// TwinCAT 3 PLC project PLC_STATE_DRIVE
// Title: PLC_STATE_DRIVE
// Author: D. Hauer
// ProjectVersion: 01.00.10
// Description: MC-PtP, NCI, Camming cyclic execution layer for motion commands
// ProgramVersion: 3.1.4024.0
// libraries:
//   Tc2_MC2, * (Beckhoff Automation GmbH)
//   Tc2_MC2_Camming, * (Beckhoff Automation GmbH)
//   Tc2_MC2_Drive, * (Beckhoff Automation GmbH)
//   Tc2_NC, * (Beckhoff Automation GmbH)
//   Tc2_Standard, * (Beckhoff Automation GmbH)
//   Tc2_System, * (Beckhoff Automation GmbH)
//   Tc2_Utilities, * (Beckhoff Automation GmbH)
//   Tc3_Module, * (Beckhoff Automation GmbH)
//   Tc2_NCI,3.3.15.0,Beckhoff Automation GmbH
//   Tc2_PlcInterpolation,3.3.18.0,Beckhoff Automation GmbH
// project tree:
//   / CAM.TcPOU, NCI.TcPOU, MAIN.TcPOU, PlcTask.TcTTO, Visualization Manager.TcVMO (not stored)
//   CAM/ FB_CamAxis.TcPOU, FB_CamCtrl.TcPOU, I_Cam_Ctrl.TcIO
//   CAM/types/ ST_CAM_CTRL.TcDUT, ST_CAM_DATA.TcDUT, ST_CAM_INFO.TcDUT, ST_CAM_READ_VALUES_PARAMETER.TcDUT (not stored), ST_CAM_STATE.TcDUT, ST_CAM_OPTIONS.TcDUT, ST_CAM_SCALING_DATA.TcDUT, ST_MOTION_FUNCTION.TcDUT (not stored), ST_MOTION_FUNCTION_POINT.TcDUT (not stored)
//   MAPPING/ MAPPING_in.TcPOU, MAPPING_out.TcPOU
//   MAPPING/types/ U_AXIS_CTRL.TcDUT (not stored), U_AXIS_NC_PARAMETER_WRT.TcDUT (not stored), U_AXIS_HOMING.TcDUT (not stored), U_AXIS_MOTION_OPTIONS.TcDUT (not stored), U_AXIS_MOVE_DATA.TcDUT (not stored), U_AXIS_GEAR_IN.TcDUT (not stored), U_AXIS_NC_PARAMETER_RD.TcDUT (not stored), U_AXIS_STATE.TcDUT (not stored), U_AXIS_INFO.TcDUT (not stored)
//   NCI/ FB_NciChannelCtrl.TcPOU, FB_NciChannel.TcPOU, I_NciChannel.TcIO, I_Nci_Ctrl.TcIO
//   NCI/types/ E_NCI_CTRL.TcDUT, E_NCI_CHANNEL_ERROR.TcDUT (not stored), E_NCI_STATE.TcDUT, E_NCI_INTERPRETER_STATE.TcDUT (not stored), ST_3D_Group.TcDUT (not stored), ST_CTRL_NCI.TcDUT, ST_NCI_M_FUNC.TcDUT, ST_Index_Group.TcDUT (not stored), ST_Interface_Group.TcDUT (not stored), ST_NciChannel_Ref.TcDUT (not stored), ST_R_Parameter.TcDUT, ST_STATE_NCI.TcDUT
//   NC_PTP/ FB_McAxisCtrl.TcPOU, FB_McAxis.TcPOU, I_McAxis.TcIO
//   NC_PTP/types/axis/ E_AxisEncoderType.TcDUT (not stored), ST_HomeParams.TcDUT
//   NC_PTP/types/control/ E_AXIS_CTRL.TcDUT, E_AXIS_STATE.TcDUT, ST_AXIS_CTRL.TcDUT, ST_AXIS_INFO.TcDUT, ST_AXIS_STATE.TcDUT, ST_GEAR_IN.TcDUT, ST_HOMING.TcDUT (not stored), ST_MOTION_OPTIONS.TcDUT, ST_MOVE_DATA.TcDUT (not stored), ST_NC_PARAMETER.TcDUT (not stored)
//   _DUT/ E_CHECK_STATE.TcDUT, E_PROGRESS.TcDUT
//   _GVL/ GlobalTextList.TcGTLO, GVL_AXIS.TcGVL, GVL_CAM.TcGVL, GVL_MSG.TcGVL, GVL_NCI.TcGVL, PLC_CONSTANT.TcGVL, PLC_VERSION.TcGVL
//   _MSG/ fb_LocalTime.TcPOU (not stored), f_MessageSet.TcPOU, MessageData.TcPOU, T_MESSAGE_LIST.TcVIS
//   _MSG/types/ e_Device.TcDUT, E_MessageType.TcDUT, E_MESSAGE_STATE.TcDUT (not stored), e_Subdevice.TcDUT, ST_Message.TcDUT
//   _UML/ CD_AXIS_ACCESS.TcCD (not stored) (excluded from build), CD_CAM_ACCESS.TcCD (not stored) (excluded from build)

CONFIGURATION PLC_STATE_DRIVE
    RESOURCE PLC ON TwinCAT3
        TASK PlcTask(INTERVAL := T#10ms, PRIORITY := 20);
        PROGRAM MAPPING_in WITH PlcTask : MAPPING_in;
        PROGRAM LEGACY WITH PlcTask : LEGACY;
        PROGRAM MAIN WITH PlcTask : MAIN;
        PROGRAM NCI WITH PlcTask : NCI;
        PROGRAM CAM WITH PlcTask : CAM;
        PROGRAM MAPPING_out WITH PlcTask : MAPPING_out;
    END_RESOURCE
END_CONFIGURATION

// ---- CAM/types/ST_CAM_CTRL.TcDUT
{attribute 'pack_mode' := '2'}
TYPE ST_CAM_CTRL :
STRUCT
  eCtrl               : E_AXIS_CTRL;    // commanded axis function
END_STRUCT
END_TYPE

// ---- CAM/types/ST_CAM_DATA.TcDUT
{attribute 'pack_mode' := '2'}
TYPE ST_CAM_DATA :
STRUCT
  // MC_CamInfo_V2 parameters
  bAtMasterPosition       : BIT;    // If AtMasterPosition is TRUE, the data related to the specified MasterPosition is determined. Otherwise the data refers to the current master position.
  nMasterIndex            : UINT;   // Index in GVL_AXIS.AxisRef[nMasterIndex]

  rMasterPosition         : LREAL;  // Master position to which the data that is determined refers. This input parameter is not necessary if AtMasterPosition is FALSE.
  rActivationPosition     : LREAL;
  nActivationMode         : UINT;
  nCamTableId             : UDINT;  // For multi-cam plate coupling, the CamTableId also has to be transferred explicitly. If a single cam plate is involved in the coupling, the CamTableId can be set to 0.
  nPointId                : UDINT;
  nNumPoints              : UDINT;  // 0 = full motion function size

  stCamScalingData        : ST_CAM_SCALING_DATA;
  stOptions               : ST_CAM_OPTIONS;
END_STRUCT
END_TYPE

// ---- CAM/types/ST_CAM_INFO.TcDUT
{attribute 'pack_mode' := '2'}
TYPE ST_CAM_INFO :
STRUCT
  bError              : BIT;
  wCamCouplingState   : ARRAY[0..7] OF WORD;
  nCamCouplingTableId : ARRAY[0..7] OF UINT;

  nNumPointsRead      : UDINT;
END_STRUCT
END_TYPE

// ---- CAM/types/ST_CAM_STATE.TcDUT
{attribute 'pack_mode' := '2'}
TYPE ST_CAM_STATE :
STRUCT
  nNumPointsRead          : UDINT;

END_STRUCT
END_TYPE

// ---- CAM/types/ST_CAM_OPTIONS.TcDUT
{attribute 'pack_mode' := '2'}
TYPE ST_CAM_OPTIONS :
STRUCT
  nInterpolationType      : UINT;
  nCamOperationMode       : UINT;
  nReferenceCamTableId    : UDINT;
END_STRUCT
END_TYPE

// ---- CAM/types/ST_CAM_SCALING_DATA.TcDUT
{attribute 'pack_mode' := '2'}
TYPE ST_CAM_SCALING_DATA :
STRUCT
  // scaling of X-axis (Master) of the CAM
  nMasterScalingMode      : UINT;
  bMasterRelative         : BOOL;
  rMasterOffset           : LREAL;
  rMasterScaling          : LREAL := 1.0;

  // scaling of Y-axis (Slave) of CAM
  nSlaveScalingMode       : UINT;
  bSlaveRelative          : BOOL;
  rSlaveOffset            : LREAL;
  rSlaveScaling           : LREAL := 1.0;
END_STRUCT
END_TYPE

// ---- NCI/types/E_NCI_CTRL.TcDUT
{attribute 'qualified_only'}
{attribute 'to_string'}
TYPE E_NCI_CTRL :
(
  NO_NCI            := -10,
  NO_AXIS_GROUP     := -2,
  NO_AXIS_INDEX     := -1,
  NO_INIT,
  INIT,
  IDLE,
  RESET,
  LOAD_PROG,
  FEED_TABLE,
  BUILD_GROUP,
  CLEAR_GROUP,

  START         := 10,
  STOP,
  STO_STOP,
  RESTART_STEP_ON,

  M_FUNC_QUIT   := 20,

  READ_R_PARA   := 30,
  WRITE_R_PARA  := 40,

  CMD_BUSY      := 100,
  CMD_DONE      := 1000,
  CMD_ERROR     := 9000
)DINT;
END_TYPE

// ---- NCI/types/E_NCI_STATE.TcDUT
{attribute 'qualified_only'}
//{attribute 'strict'}
{attribute 'to_string'}
TYPE E_NCI_STATE :
(
  NO_NCI            := -10,
  NO_AXIS_GROUP     := -2,
  NO_AXIS_INDEX     := -1,
  NO_INIT,
  INIT,
  IDLE,
  RESET,
  LOAD_PROG,
  FEED_TABLE,
  BUILD_GROUP,
  CLEAR_GROUP,

  START         := 10,
  STOP,
  STO_STOP,
  RESTART_STEP_ON,

  M_FUNC_QUIT   := 20,

  READ_R_PARA   := 30,
  WRITE_R_PARA  := 40

)DINT;
END_TYPE

// ---- NCI/types/ST_CTRL_NCI.TcDUT
{attribute 'pack_mode' := '2'}
TYPE ST_CTRL_NCI :
STRUCT
  eCmd        : E_NCI_CTRL := E_NCI_CTRL.INIT;
  rOverride   : REAL := 47.11;

END_STRUCT
END_TYPE

// ---- NCI/types/ST_NCI_M_FUNC.TcDUT
{attribute 'pack_mode' := '2'}
TYPE ST_NCI_M_FUNC :
STRUCT
  FastMFuncMask   : ARRAY [1..5] OF DWORD;
  HskMFuncNo      : UINT;
  HskMFuncReq     : WORD;
  HFuncValue      : UDINT; 
END_STRUCT
END_TYPE

// ---- NCI/types/ST_R_Parameter.TcDUT
{attribute 'pack_mode' := '2'}
TYPE ST_R_Parameter :
STRUCT
  _nStart               : DINT := 901;
  _nCount               : DINT :=   4;
  _rRParamsWrite        : ARRAY[0..MAX_R_PARA] OF LREAL := [11.11, 22.22, 33.33, 456.22];
  _rRParamsRead         : ARRAY[0..MAX_R_PARA] OF LREAL;
END_STRUCT
END_TYPE

// ---- NCI/types/ST_STATE_NCI.TcDUT
{attribute 'pack_mode' := '2'}
TYPE ST_STATE_NCI :
STRUCT
  eState        : E_NCI_STATE; // eCmd with offsets E_PROGRESS

  bMFuncReq     : BIT;  // M function request is active from channel

  nMFunc        : WORD; // number of active M function

  nItpState     : UINT; 
                         (*  Interpreter Operation State:
                            0  = Init failed
                            1  = Idle
                            2  = Ready
                            3  = Started
                            4  = Scanning
                            5  = Running
                            6  = Stay running
                            7  = Write table
                            8  = Search line
                            9  = End
                            10 = Single Step
                            11 = Aborting
                            12 = Aborted
                            13 = Fault
                            14 = Reset
                            15 = Stop
                            16 = Wait function
                            17 = Flush buffers
                          *) 

  rAxisOverride : REAL; // active override in cyclic NCI interface

END_STRUCT
END_TYPE

// ---- NC_PTP/types/axis/ST_HomeParams.TcDUT
TYPE ST_HomeParams :
STRUCT
  Position              : LREAL;
  HomingMode            : Tc2_MC2.MC_HomingMode;
  Options               : Tc2_MC2.ST_HomingOptions;

  InvertHomeSensor      : BIT := FALSE;   //Set to true,  NormallyClosed home sensor
  SimulateHomeSensor    : BIT := FALSE;   //Set to true,  homed on encoder index only. The homing methode 'hardware sync' must be used then.

  UseLimitMin           : BIT := TRUE;    //Set to false, no negative limit sensor.

  InvertLimitMin        : BIT := FALSE;   //Set to true,  NC negative limit sensor
  HomeOnLimitMin        : BIT := FALSE;   //Set to true,  homed on negative limit sensor 

  UseLimitMax           : BIT := TRUE;    //Set to false, no positive limit sensor.

  InvertLimitMax        : BIT := FALSE;   //Set to true,  NC positive limit sensor
  HomeOnLimitMax        : BIT := FALSE;   //Set to true,  homed on positive limit sensor 
  
  // It is not allowed to use more than 1 of the 3 switches: SimulateHomeSensor, HomeOnLimitMin, HomeOnLimitMax
  
END_STRUCT
END_TYPE

// ---- NC_PTP/types/control/E_AXIS_CTRL.TcDUT
{attribute 'qualified_only'}
{attribute 'strict'}
{attribute 'to_string'}
TYPE E_AXIS_CTRL :
(
  AXIS_NULL,   // null command
  AXIS_INIT,
  AXIS_DISABLE,
  AXIS_ENABLE,

  AXIS_IDLE     := 10, // clear axis and enable
  AXIS_HOME,
  AXIS_MOVE_POS,
  AXIS_MOVE_VELO,
  AXIS_HALT,
  AXIS_STOP,

  AXIS_RESET              := 19,
  AXIS_STARTUP            := 20,

  AXIS_MOVE_BUFFER        := 30,
  AXIS_MOVE_BUFFER_VELO,

  AXIS_PARAMETER_READ     := 40, // command for reading and writing parameter
  AXIS_PARAMETER_WRITE,
  AXIS_PARAMETER_WRITE_PERSISTENT,


  AXIS_GEAR_IN            := 50,
  AXIS_GEAR_OUT,
  AXIS_GEAR_IN_MULTIMASTER,

  CAM_INIT                := 60,
  CAM_IN,
  CAM_SCALING,
  CAM_INFO,
  CAM_RD_MOTION_FUNCTION,
  CAM_RD_MOTION_FUNCTION_POINT,
  CAM_RD_MOTION_FUNCTIONS_VALUES,
  CAM_WRT_MOTION_FUNCTION,
  CAM_WRT_MOTION_FUNCTION_POINT

)UINT;
END_TYPE

// ---- NC_PTP/types/control/E_AXIS_STATE.TcDUT
{attribute 'qualified_only'}
{attribute 'to_string'}
TYPE E_AXIS_STATE :
(
  AXIS_NULL,   // null reaction to command
  AXIS_INIT,
  AXIS_DISABLE,
  AXIS_ENABLE,

  AXIS_NO_INIT  := 9,
  
  AXIS_IDLE     := 10, // clear axis and enable
  AXIS_HOME,
  AXIS_MOVE_POS,
  AXIS_MOVE_VELO,
  AXIS_HALT,
  AXIS_STOP,

  AXIS_RESET              := 19,
  AXIS_STARTUP            := 20,

  AXIS_MOVE_BUFFER        := 30,
  AXIS_MOVE_BUFFER_VELO,

  AXIS_PARAMETER_READ     := 40, // command for reading and writing parameter
  AXIS_PARAMETER_WRITE,
  AXIS_PARAMETER_WRITE_PERSISTENT,


  AXIS_GEAR_IN            := 50,
  AXIS_GEAR_OUT,
  AXIS_GEAR_IN_MULTIMASTER,

  CAM_INIT                := 60,
  CAM_IN,
  CAM_SCALING,
  CAM_INFO,
  CAM_RD_MOTION_FUNCTION,
  CAM_RD_MOTION_FUNCTION_POINT,
  CAM_RD_MOTION_FUNCTIONS_VALUES,
  CAM_WRT_MOTION_FUNCTION,
  CAM_WRT_MOTION_FUNCTION_POINT

)UINT;
END_TYPE

// ---- NC_PTP/types/control/ST_AXIS_CTRL.TcDUT
{attribute 'pack_mode' := '2'}
TYPE ST_AXIS_CTRL :
STRUCT
  eCtrl               : E_AXIS_CTRL;    // commanded axis function
  eProgress           : E_PROGRESS;     // progress command for synced functions
END_STRUCT
END_TYPE

// ---- NC_PTP/types/control/ST_AXIS_INFO.TcDUT
{attribute 'pack_mode' := '2'}
TYPE ST_AXIS_INFO :
STRUCT
  bEnabled    : BIT; // Enabled: check if ControlLoop is closed and active
  bReferenced : BIT; // Axis homing bit
  bReady      : BIT; // enabled & NOT bError & no Axis Function requested
  bBusy       : BIT; // axis function requested or active
  bError      : BIT;
  bTimeout    : BIT; // for move cmds or switching drive on timeout
  bInTarget   : BIT; // ActPos = SetPos --> position check is done with configured window in NC
  bStandstill : BIT; // No Error and NOT moving
 
  nErrorId            : UDINT;

  rActPos             : LREAL;
  rActVelo            : LREAL;
  rPosDiff            : LREAL;

  dwCoupleState       : DWORD;   // cyclic information about axis couple state
END_STRUCT
END_TYPE

// ---- NC_PTP/types/control/ST_AXIS_STATE.TcDUT
{attribute 'pack_mode' := '2'}
TYPE ST_AXIS_STATE :
STRUCT
  eState        : E_AXIS_STATE; // mirror the requested command + E_PROGRESS
  eAxisEncoder  : E_AxisEncoderType;
END_STRUCT
END_TYPE

// ---- NC_PTP/types/control/ST_GEAR_IN.TcDUT
{attribute 'pack_mode' := '2'}
TYPE ST_GEAR_IN :
STRUCT  
  nAxisIndexMaster    : ARRAY [1..4] OF BYTE; // Index of Master1-4
  rGearRatio          : ARRAY [1..4] OF REAL; 
  Acceleration        : REAL;
  Deceleration        : REAL;
  Jerk                : REAL;  
END_STRUCT
END_TYPE

// ---- NC_PTP/types/control/ST_MOTION_OPTIONS.TcDUT
{attribute 'pack_mode' := '2'}
TYPE ST_MOTION_OPTIONS :
STRUCT
  eBufferMode   : Tc2_MC2.MC_BufferMode;

END_STRUCT
END_TYPE

// ---- _DUT/E_CHECK_STATE.TcDUT
{attribute 'qualified_only'}
{attribute 'strict'}
{attribute 'to_string'}
TYPE E_CHECK_STATE :
(
  CHECK_INIT,
  AXIS_INDEX_OUT_OF_RANGE         :=  10,

	AXIS_REF_POINTER_INVALID        := 100,
  AXIS_CTRL_POINTER_INVALID,
  AXIS_STATE_POINTER_INVALID,
  AXIS_INFO_POINTER_INVALID,
  AXIS_DATA_POINTER_INVALID,
  AXIS_NC_PARAMETER_POINTER_INVALID,
  AXIS_HOME_PARAMETER_POINTER_INVALID,
  AXIS_GEAR_IN_PARAMETER_POINTER_INVALID,
  AXIS_GEAR_IN_MULTIMASTER_POINTER_INVALID,
  AXIS_MOTION_OPTIONS_POINTER_INVALID,

  NCI_NOT_ACTIVATED               := 200,
  NCI_CHANNEL_REF_POINTER_INVALID,
  NCI_AXIS_CONFIG_POINTER_INVALID,
  NCI_MCS_AXIS_POINTER_INVALID,
  NCI_AUX_AXIS_POINTER_INVALID,
  NCI_CTRL_POINTER_INVALID,
  NCI_STATE_POINTER_INVALID,
  NCI_R_PARAMETER_READ_POINTER_INVALID,
  NCI_R_PARAMETER_wRITE_POINTER_INVALID,
  NCI_M_FUNC_POINTER_INVALID,

  CAM_NOT_ACTIVATED               := 300,
  CAM_SLAVE_AXIS_REF_INVALID,
  CAM_SLAVE_ITF_MC_AXIS_INVALID,
  CAM_MASTER_AXIS_REF_INVALID,
  CAM_MOTION_FUNCTION_POINTER_INVALID,
  CAM_MOTION_FUNCTION_POINT_POINTER_INVALID,

  CHECK_DONE                      := 10000
  
)UINT;
END_TYPE

// ---- _DUT/E_PROGRESS.TcDUT
{attribute 'qualified_only'}
//{attribute 'strict'}
{attribute 'to_string'}
TYPE E_PROGRESS :
(
  // progress is used in project to mirror state of requested command/function
  INVALID,
  INIT,
	BUSY          :=  100,
  STARTUP       :=  200,
  PREPARE       :=  300,
  READY         :=  400,
  WAITING       :=  500,
  WORKING       :=  600,
  FINISHING     :=  700,

  DONE          := 1000,

  NOT_EXIST     := 6000,
  ERROR         := 9000

)UINT;
END_TYPE

// ---- _MSG/types/e_Device.TcDUT
{attribute 'to_string'}
TYPE e_Device :
(
  Device_Null,
  General           :=   100,

  CaGroup           :=   200,
  Xpu               :=   300,
  XpuCtrl           :=   400,

  Mover             :=   500,
  MoverCtrl         :=   600,

  XtsTransportUnit  :=   700,

  XtsStation        :=  1000,


  Camming           :=  3000,
  NciChannel        :=  4000,
  NciChannelCtrl    :=  5000,
  Axis              :=  7000,
  Data              := 10000
)DINT;
END_TYPE

// ---- _MSG/types/E_MessageType.TcDUT
{attribute 'strict'}
{attribute 'to_string'}
TYPE E_MessageType :
(
  eMessageEmpty,
  eMessageInfo,
  eMessageWarn,
  eMessageError
)DINT;
END_TYPE

// ---- _MSG/types/e_Subdevice.TcDUT
{attribute 'strict'}
{attribute 'to_string'}
TYPE e_Subdevice :
(
  SubDevice_Null,
  // Motion Control FB Instances
  fbPowerOn               := 10,
  fbPowerOff,
  fbReset,
  fbResetSercos,
  fbHalt,
  fbStop,
  fbHome,
  fbJog,
  fbMoveToPosition,
  fbMoveVelo,
  fbMoveVelocity1,
  fbMoveVelocity2,
  fbMoveAbsolute1,
  fbMoveAbsolute2,
  fbMoveEndless,
  fbMovePtP,


  // CA CollisionAvoidance FB instances
  // CA group fb instances
  fbCaGroup             := 30,
  fbMoveToPosCa,
  fbSendToAbsPosCa,
  fbSendToModuloPosCa,
  fbGearInPosCa,
  fbGroupAddAxis,
  fbGroupRemoveAxis,
  fbGroupDisable,
  fbGroupEnable,
  fbGroupErrorRead,
  fbGroupStatusRead,
  fbGroupReset,
  fbGroupStop,

  fbGearIn              := 50,
  fbGearOut,
  fbGearInMultiMaster,

  fbCamOut              := 80,
  fbCamInV2,
  fbCamScalingV2,
  fbCamInfoV2,
  fbReadMotionFunction,
  fbReadMotionFunctionPoint,
  fbReadMotionFunctionValues,
  fbWriteMotionFunction,
  fbWriteMotionFunctionPoint,
  fbSetOnlineChangeMode,

  fbReadParameter       := 100,
  fbReadBoolParameter,
  fbWriteParameter,
  fbWriteBoolParameter,
  fbWriteParameterPersistent,



	fbBuildGroup          := 200,
	fbClearGroup,
	fbLoadProg,
	fbResetItp,
	fbStartStopItp,
	fbEStopItp,
	fbStepOnAfterEStopItp,
	fbConfirmHskItp,
	fbDelDtgItp,
	fbNciFeedTablePreparation,
	fbNciFeedTable,
	fbReadLine,
  fbItpReadRParams,
  fbItpWriteRParams,
  Get_ItpState,
  Get_Error,

  AxisControl           := 1000,
  AxisStartUp,
  AxisCycle,
  AxisIdle,

  NciControl           := 2000,
  NciStartUp,
  NciCycle,
  NciIdle,

  StationLinkedList     := 3000,
  StationInitList,
  StationAddHead,
  StationAddTail,
  StationGetHead,
  StationRemoveHeadValue,

  StationControl        := 4000,
  StationState, 

  Xpu_fbEnvironment     := 5000,
  Xpu_fbProcessingUnit,
  Xpu_fbXpuPart,
  Xpu_fbXpuTrack,
  Xpu_fbMc2CaGroup,

  Xpu_fbPartModules     := 5500,

  Xpu_fbMoverXpu        := 6000,

  CamControl            := 8000,
  CamStartUp,
  CamCycle
)DINT;
END_TYPE

// ---- _MSG/types/ST_Message.TcDUT
TYPE ST_Message :
STRUCT
  eType         : e_MessageType;
  eDevice       : e_Device;
  eSubdevice    : e_SubDevice;
  {attribute 'displaymode':='hex'}
  iErrorNumber  : LINT;
  tTime         : STRING(24);
  sText         : STRING(256);
END_STRUCT
END_TYPE

// ---- _GVL/GVL_AXIS.TcGVL
{attribute 'qualified_only'}
VAR_GLOBAL

  AxisRef                     : ARRAY[1..PLC_CONSTANT.MAX_AXIS] OF Tc2_MC2.AXIS_REF;

  Control                     : ARRAY[1..PLC_CONSTANT.MAX_AXIS] OF FB_McAxisCtrl;     // cyclic interface for accepting and executing orders
  Ctrl                        : ARRAY[1..PLC_CONSTANT.MAX_AXIS] OF ST_AXIS_CTRL;      // command structure to write into
  State                       : ARRAY[1..PLC_CONSTANT.MAX_AXIS] OF ST_AXIS_STATE;     // state structure to read from
  Info                        : ARRAY[1..PLC_CONSTANT.MAX_AXIS] OF ST_AXIS_INFO;      // axis state and position data to read from
  Data                        : ARRAY[1..PLC_CONSTANT.MAX_AXIS] OF ST_MOVE_DATA;      // axis data to write into

  NcParameterWrt              : ARRAY[1..PLC_CONSTANT.MAX_AXIS] OF ST_NC_PARAMETER;   // struct for a single parameter value put/get your data here before/after using Ctrl
  NcParameterRd               : ARRAY[1..PLC_CONSTANT.MAX_AXIS] OF ST_NC_PARAMETER;   // struct for a single parameter value put/get your data here before/after using Ctrl

  HomeParameter               : ARRAY[1..PLC_CONSTANT.MAX_AXIS] OF ST_HOMING;         // homing parameter for each axis

  GearInParameter             : ARRAY[1..PLC_CONSTANT.MAX_AXIS] OF ST_GEAR_IN;        // GearIn and GearInMultiMaster, index to master axes[1-4], rGearRatio[1-4]

  MotionOptions               : ARRAY[1..PLC_CONSTANT.MAX_AXIS] OF ST_MOTION_OPTIONS; // additional motion parameters
END_VAR

// ---- _GVL/GVL_CAM.TcGVL
{attribute 'qualified_only'}
VAR_GLOBAL
  //-----------------------------------------------------------------------------
  // command and state structure
  //  - datafields for anyone to access
  //    - ADS via symbol
  //    - cyclic mapping to any other cyclic network/runtime
  //-----------------------------------------------------------------------------
  Ctrl                        : ARRAY[1..PLC_CONSTANT.MAX_AXIS] OF ST_CAM_CTRL;      // command structure to write into
  State                       : ARRAY[1..PLC_CONSTANT.MAX_AXIS] OF ST_CAM_STATE;     // state structure to read from


  //-----------------------------------------------------------------------------
  // data and info structure
  //  - parameter data fields for
  //    - Ctrl  --> Data
  //    - State --> Info
  //-----------------------------------------------------------------------------
  Info                        : ARRAY[1..PLC_CONSTANT.MAX_AXIS] OF ST_CAM_INFO;
  Data                        : ARRAY[1..PLC_CONSTANT.MAX_AXIS] OF ST_CAM_DATA;


  //-----------------------------------------------------------------------------
  // R/W datafields
  // - get your data here after read
  // - put your data here before write
  //
  //    - Motion Function
  //    - Motion Function Point
  //-----------------------------------------------------------------------------
  MotionFunction              : ARRAY[1..PLC_CONSTANT.MAX_AXIS] OF ST_MOTION_FUNCTION;
  MotionFunctionPoint         : ARRAY[1..PLC_CONSTANT.MAX_AXIS] OF ST_MOTION_FUNCTION_POINT;


  //-----------------------------------------------------------------------------
  // cyclic interface function block: FB_CamCtrl
  //  - MC_Camming functions are here 
  //-----------------------------------------------------------------------------
{IF defined (CAM)}
  Control                     : ARRAY[1..PLC_CONSTANT.MAX_AXIS] OF FB_CamCtrl;
{ELSE}
  Control                     : ARRAY[1..PLC_CONSTANT.MAX_AXIS] OF I_Cam_Ctrl;
{END_IF}
END_VAR

// ---- _GVL/GVL_MSG.TcGVL
{attribute 'qualified_only'}
VAR_GLOBAL CONSTANT
  //-----------------------------------------------------------------------------
  // file paths for message system
  //  - compiler define option WIN switches to Windows file paths
  //-----------------------------------------------------------------------------
{IF NOT defined (BSD)}
  {info 'WIN folders'}
  LOG_DIR               : STRING  := 'C:\TwinCAT\#MsgFiles\';
{ELSE}
  {info 'BSD folders'}
  LOG_DIR               : STRING  := '/usr/local/etc/TwinCAT/#MsgFiles/';
{END_IF}

  LOG_FILE              : STRING  := 'MSG_PLCSD_';

  MAX_MESSAGE           : UINT     := 200; // max entry in message list
END_VAR
VAR_GLOBAL

  // diag data
  dbg_AxisIdxGearIn               : ARRAY[1..PLC_CONSTANT.MAX_AXIS]      OF BYTE; // diag for Axis gear in
  
  dbg_AxisIdxGearInMultiMaster    : ARRAY[1..PLC_CONSTANT.MAX_AXIS,1..4] OF BYTE; // diag for Axis gear in multi master
  
  dbg_AxisIdxCamIn                : ARRAY[1..PLC_CONSTANT.MAX_AXIS]      OF BYTE; // diag for Axis cam in


  Messages                        : ARRAY[1..MAX_MESSAGE] OF ST_Message;
  MessageIndex                    : UINT := 0; // message index
  MessageError                    : UINT := 0; // error counter

  fbLocalTime                     : fb_LocalTime;
  dtLocalTime                     : DT;
  sLocalTime                      : STRING;

  MessageLevelAxisPtp             : ARRAY[1..PLC_CONSTANT.MAX_AXIS]   OF E_MessageType;
  MessageLevelAxisCam             : ARRAY[1..PLC_CONSTANT.MAX_AXIS]   OF E_MessageType;
  MessageLevelNciChn              : ARRAY[1..PLC_CONSTANT.MAX_NCI_CH] OF E_MessageType;

{IF defined (TEST)}
  {info 'TEST logging enabled'}
  MessageLevel                    : E_MessageType := eMessageVerbose; // a lot of messages
{ELSE}
  MessageLevel                    : E_MessageType := eMessageError;    // not as much messages 
{END_IF}

END_VAR

// ---- _GVL/GVL_NCI.TcGVL
{attribute 'qualified_only'}
VAR_GLOBAL
  stAxisConfig                : ARRAY[1..MAX_NCI_CH] OF ST_3D_Group;     // NC Axis Id to build NCI group

  stChannelCtrl               : ARRAY[1..MAX_NCI_CH] OF ST_CTRL_NCI;
  stChannelState              : ARRAY[1..MAX_NCI_CH] OF ST_STATE_NCI;

  sProgName                   : ARRAY[1..MAX_NCI_CH] OF STRING(255):= ['/usr/local/etc/TwinCAT/Mc/Nci/Test_GST.nc'];
  sProgNameActive             : ARRAY[1..MAX_NCI_CH] OF STRING(255);

  R_ParameterRead             : ARRAY[1..MAX_NCI_CH] OF ST_R_Parameter;
  R_ParameterWrite            : ARRAY[1..MAX_NCI_CH] OF ST_R_Parameter;

  M_FunctionCyclic            : ARRAY[1..MAX_NCI_CH] OF ST_NCI_M_FUNC; // scope variable for M function tests

{IF defined (NCI)}
  fbNciCtrl                   : ARRAY[1..MAX_NCI_CH] OF FB_NciChannelCtrl;
{ELSE}
  fbNciCtrl                   : ARRAY[1..MAX_NCI_CH] OF I_Nci_Ctrl;
{END_IF}
END_VAR

// ---- _GVL/PLC_CONSTANT.TcGVL
//{attribute 'qualified_only'}
VAR_GLOBAL CONSTANT


  //-----------------------------------------------------------------------------
  // AXIS related limits
  //-----------------------------------------------------------------------------
  MAX_AXIS              : UINT    := 3;
  MAX_RETRY             : UINT    := 5;


  //-----------------------------------------------------------------------------
  // NCI related limits and *.nc standard folder
  //-----------------------------------------------------------------------------
{IF NOT defined (BSD)}
  NCI_DIR               : STRING  := 'C:\TwinCAT\Mc\Nci\';
{ELSE}
  NCI_DIR               : STRING  := '/usr/local/etc/TwinCAT/Mc/Nci/';
{END_IF}

{IF defined (NCI)}
  {info 'NCI Channel active'}
  NCI_ACTIVE            : BOOL    := TRUE;
  CONFIG_NAME           : STRING  := 'NCI_Spec_Ch_';
{ELSE}
  {info 'NCI Channel NOT active'}
  NCI_ACTIVE            : BOOL    := FALSE;
  CONFIG_NAME           : STRING  := 'NCI_NOT_ACTIVE';
{END_IF}

  MAX_NCI_CH            : UINT    := 1;

  MAX_PATH_STEPS        : UINT    := 5;
  MAX_MC_AXIS           : UINT    := 3;
  MAX_AUX_AXIS          : UINT    := 2;
  MAX_R_PARA            : UINT    := 10;


  //-----------------------------------------------------------------------------
  // CAMMING related limits
  //-----------------------------------------------------------------------------
{IF defined (CAM)}
  {info 'CAMMING active'}
  CAM_ACTIVE                  : BOOL    := TRUE;
{ELSE}
  {info 'CAMMING NOT active'}
  CAM_ACTIVE                  : BOOL    := FALSE;
{END_IF}

  MAX_CAM_CH                  : UINT    := 1;

  MAX_MOTION_FUNCTION_POINTS  : UINT    := 10;

END_VAR

// ---- _GVL/PLC_VERSION.TcGVL
{attribute 'qualified_only'}
VAR_GLOBAL CONSTANT
  VERSION               : STRING := 'V 01.00.10';

  // 2024 06 10 HAUD
  //
  // - TC_PLC_MOTION_LAYER: 
  //    - rename repository
  //    - remove LEGACY compatibility
  //
  // - PLC_OPEN_DRIVE:
  //    - deprecated


  // 2024 05 31 HAUD
  // 
  // V 01.00.02
  // precompiler defines: 
  //  - BSD: 
  //    - Tc-BSD file system is used else Windows file system is used
  //
  //  - TEST:
  //    - GVL_MSG.MessageLevel
  // Axis, Cam, Nci have individual message levels now

  // 2024 03 09 HAUD
  // 
  // V 01.00.01
  // MC PtP - execution layer with optional mapping
  // NCI    - execution layer with optional mapping
  // CAM    . execution layer with optional mapping
  // precompiler defines: 
  //  - WIN: windows file system is used else Tc-BSD file system is used
  //  - NCI: NCI libraries are linked in project
  //  - CAM: Camming libraries are linked in project
  //  - AXIS_MAP: mapping is used


  // 2024 02 15 HAUD
  // 
  // V 00.50.04
  //
  // Buffered moves test
  // CamIn Test --> TODO MultiCam
  // Message system, cyclic check for write
  

  // 2024 01 12 HAUD
  //
  // V 00.50.03
  //
  // Building is done
  // start of UnitTesting

  // 2024 01 17 HAUD
  //
  // V 00.50.02
  // 
  // start camming implementation (MC_CamIn_V2)
  // legacy namespace available for downward compatibility of ADS Symbol names

  // 2023 12 23 HAUD
  // NC_PTP
  // - redesign for PLC_OPEN_DRIVE started 
  //    --> E_PROGRESS for state feedback
  // - FB_AxisControl inherits FB_McAxis


  //  2023 10 19
  //  HAUD
  // first draft 
  // TODO: everything

END_VAR

// ---- CAM/I_Cam_Ctrl.TcIO
INTERFACE I_Cam_Ctrl

PROPERTY Axes : reference TO ARRAY[1..PLC_CONSTANT.MAX_AXIS] OF AXIS_REF
SET
END_SET
END_PROPERTY

PROPERTY AxisCtrl : pointer to ARRAY[1..PLC_CONSTANT.MAX_AXIS] OF st_axis_ctrl
SET
END_SET
END_PROPERTY

PROPERTY AxisData : pointer to ARRAY[1..PLC_CONSTANT.MAX_AXIS] OF ST_CAM_DATA
SET
END_SET
END_PROPERTY

PROPERTY AxisIndex : uint
SET
END_SET
END_PROPERTY

PROPERTY AxisInfo : pointer to ARRAY[1..PLC_CONSTANT.MAX_AXIS] OF ST_AXIS_INFO
SET
END_SET
END_PROPERTY

PROPERTY AxisState : pointer to ARRAY[1..PLC_CONSTANT.MAX_AXIS] OF ST_CAM_STATE
SET
END_SET
END_PROPERTY

METHOD Cycle  : e_progress
END_METHOD

PROPERTY ItfMcAxes : array[1..MAX_AXIS] of I_McAxis
SET
END_SET
END_PROPERTY

PROPERTY MotionFunction : POINTER TO ARRAY[1..MAX_AXIS] OF ST_MOTION_FUNCTION
SET
END_SET
END_PROPERTY

PROPERTY MotionFunctionPoint : pointer to array[1..MAX_AXIS] of ST_MOTION_FUNCTION_POINT
SET
END_SET
END_PROPERTY

END_INTERFACE

// ---- NCI/I_NciChannel.TcIO
INTERFACE I_NciChannel

METHOD BuilDGroup : E_PROGRESS
VAR_INPUT
  Execute           : BOOL;
END_VAR
END_METHOD

PROPERTY CfgAxes : POINTER TO ST_3D_Group
SET
END_SET
END_PROPERTY

PROPERTY ChannelRef : POINTER TO ST_NciChannel_Ref
SET
END_SET
END_PROPERTY

METHOD ClearGroup : E_PROGRESS
VAR_INPUT
  Execute           : BOOL;
END_VAR
END_METHOD

METHOD ConfirmHSK : E_PROGRESS
VAR_INPUT
  Execute           : BOOL;
END_VAR
END_METHOD

METHOD DeleteDistanceToGo : E_PROGRESS
VAR_INPUT
  Execute           : BOOL;
END_VAR
END_METHOD

(*
===============================================================
Error-Flag
===============================================================
*)
PROPERTY Error : BOOL
GET
END_GET
END_PROPERTY

METHOD Error_Get : BOOL
END_METHOD

METHOD EStop : E_PROGRESS
VAR_INPUT
  Execute           : BOOL;
END_VAR
END_METHOD

METHOD GetChannelOverride : real
VAR_INPUT
END_VAR
END_METHOD

METHOD GetItpState : uint
VAR_INPUT
END_VAR
END_METHOD

METHOD GetLoadedProg : string
VAR_INPUT
END_VAR
END_METHOD

(*
===============================================================
Handshake: Announce and acknowledge M-Functions
===============================================================
*)
PROPERTY HSK : BOOL
GET
END_GET
END_PROPERTY

PROPERTY ItpAxes : ST_3D_Group
GET
END_GET
END_PROPERTY

METHOD ItpReset   : E_PROGRESS
VAR_INPUT
  Execute           : BOOL;
END_VAR
END_METHOD

METHOD LoadProg   : E_PROGRESS
VAR_INPUT
  Execute           : BOOL;
END_VAR
END_METHOD

PROPERTY M_FuncReq : word
GET
END_GET
END_PROPERTY

(*
===============================================================
M-Function
===============================================================
*)
PROPERTY MFunc : INT
GET
END_GET
END_PROPERTY

PROPERTY Override : LREAL
GET
END_GET
SET
END_SET
END_PROPERTY

(*
===============================================================
actual path velo [Units/s]
===============================================================
*)
PROPERTY PathVelo : LREAL
GET
END_GET
END_PROPERTY

(*
===============================================================
G-Code Program Name (sFilePath)
===============================================================
*)
PROPERTY Prog : STRING(255)
GET
END_GET
SET
END_SET
END_PROPERTY

PROPERTY R_ParameterRead : Pointer to ST_R_Parameter;
SET
END_SET
END_PROPERTY

PROPERTY R_ParameterWrite : pointer to ST_R_Parameter;
SET
END_SET
END_PROPERTY

METHOD ReadLine   : E_PROGRESS
VAR_INPUT
  Execute           : BOOL;
END_VAR
//Read G-Code actual Line
VAR_OUTPUT
  ActProgLine       : STRING(100);
END_VAR
END_METHOD

METHOD ReadRParams : E_PROGRESS
VAR_INPUT
  Execute  : BOOL;
END_VAR
END_METHOD

METHOD StartStop : E_PROGRESS
VAR_INPUT
  Execute           : BOOL;
  Start             : BOOL;
  Stop              : BOOL;
END_VAR
END_METHOD

METHOD StepOnAfterEStop : E_PROGRESS
VAR_INPUT
  Execute: BOOL;
END_VAR
END_METHOD

METHOD WriteRParams : E_PROGRESS
VAR_INPUT
  Execute : BOOL;
END_VAR
END_METHOD

END_INTERFACE

// ---- NCI/I_Nci_Ctrl.TcIO
INTERFACE I_Nci_Ctrl

METHOD Cycle : E_PROGRESS
VAR_INPUT
END_VAR
END_METHOD

END_INTERFACE

// ---- NC_PTP/I_McAxis.TcIO
INTERFACE I_McAxis

METHOD Disable : E_PROGRESS
VAR_INPUT
  Execute           : BOOL;
END_VAR
END_METHOD

METHOD Enable : E_PROGRESS
VAR_INPUT
  Execute           : BOOL;
END_VAR
END_METHOD

METHOD Halt : E_PROGRESS
VAR_INPUT
  Execute           : BOOL;
  Dec               : LREAL;
  Jerk              : LREAL;
END_VAR
END_METHOD

METHOD Reset : E_PROGRESS
VAR_INPUT
  Execute           : BOOL;
END_VAR
END_METHOD

METHOD Stop : E_PROGRESS
VAR_INPUT
  Execute           : BOOL;
  Dec               : LREAL;
  Jerk              : LREAL;
END_VAR
END_METHOD

END_INTERFACE

// ---- MAPPING/MAPPING_in.TcPOU
PROGRAM MAPPING_in
VAR CONSTANT
{IF defined (AXIS_MAP)}
  {info 'MAPPING_in - ACTIVE'}
  bBypassMapping    : BOOL  := FALSE;
{ELSE}
  bBypassMapping    : BOOL  := TRUE;
{END_IF}
END_VAR
VAR
{IF defined (AXIS_MAP)}
  AxisCTrl          : U_AXIS_CTRL;
  AxisMoveData      : U_AXIS_MOVE_DATA;
  AxisMotionOptions : U_AXIS_MOTION_OPTIONS;

  AxisGearInData    : U_AXIS_GEAR_IN;
  AxisHoming        : U_AXIS_HOMING;
  AxisParameterWrt  : U_AXIS_NC_PARAMETER_WRT;
  
{ELSE}
  AxisCTrl          : BYTE;
  AxisMoveData      : BYTE;
  AxisMotionOptions : BYTE;

  AxisGearInData    : BYTE;
  AxisHoming        : BYTE;
  AxisParameterWrt  : BYTE;
{END_IF}

  szAxisPara,
  szAxisHoming,
  szAxisGearData,
  szAxisMotionOptions,
  szAxisMoveData,
  szAxisCtrl        : ARRAY[1..2] OF UDINT;


END_VAR


szAxisCtrl[1]           := SIZEOF(AxisCTrl);
szAxisCtrl[2]           := SIZEOF(GVL_AXIS.Ctrl);

szAxisMoveData [1]      := SIZEOF(AxisMoveData);
szAxisMoveData [2]      := SIZEOF(GVL_AXIS.Data);

szAxisMotionOptions [1] := SIZEOF(AxisMotionOptions);
szAxisMotionOptions [2] := SIZEOF(GVL_AXIS.MotionOptions);

szAxisGearData [1]      := SIZEOF(AxisGearInData);
szAxisGearData [2]      := SIZEOF(GVL_AXIS.GearInParameter);

szAxisHoming [1]        := SIZEOF(AxisHoming);
szAxisHoming [2]        := SIZEOF(GVL_AXIS.HomeParameter);

szAxisPara [1]          := SIZEOF(AxisParameterWrt);
szAxisPara [2]          := SIZEOF(GVL_AXIS.NcParameterWrt);



IF bBypassMapping 
THEN 
  RETURN; 
END_IF


memcpy(ADR(GVL_AXIS.Ctrl),            ADR(AxisCtrl),           SIZEOF(AxisCTrl));
memcpy(ADR(GVL_AXIS.Data),            ADR(AxisMoveData),       SIZEOF(AxisMoveData));
memcpy(ADR(GVL_AXIS.MotionOptions),   ADR(AxisMotionOptions),  SIZEOF(AxisMotionOptions));

memcpy(ADR(GVL_AXIS.GearInParameter), ADR(AxisGearInData),     SIZEOF(AxisGearInData));
memcpy(ADR(GVL_AXIS.HomeParameter),   ADR(AxisHoming),         SIZEOF(AxisHoming));
memcpy(ADR(GVL_AXIS.NcParameterWrt),  ADR(AxisParameterWrt),   SIZEOF(AxisParameterWrt));

END_PROGRAM

// ---- MAIN.TcPOU
PROGRAM MAIN
VAR
  bInit                     : BOOL;
  eInit                     : E_PROGRESS;

  nAxis,
  nAxisInit                 : UINT;

  stMsg                     : ST_Message;

  tWriteLog                 : TIME := T#10S;
  tonWriteLog               : Tc2_Standard.TON;
END_VAR

//-----------------------------------------------------------------------------------------------------------------
// Local time; used for timestamps
//-----------------------------------------------------------------------------------------------------------------
GVL_MSG.fbLocalTime(
                    sLocalTime                => GVL_MSG.sLocalTime, 
                    dtLocalTime               => GVL_MSG.dtLocalTime);
//-----------------------------------------------------------------------------------------------------------------
//-----------------------------------------------------------------------------------------------------------------
// /assign dataflow
//-----------------------------------------------------------------------------------------------------------------
FOR nAxis := 1 TO PLC_CONSTANT.MAX_AXIS
DO
  GVL_AXIS.Control[nAxis].AxisIndex           := nAxis;
  GVL_AXIS.Control[nAxis].MessageLevel        := GVL_MSG.MessageLevelAxisPtp[nAxis];

  GVL_AXIS.Control[nAxis].AxisCtrl            := ADR(GVL_AXIS.Ctrl);          // command
  GVL_AXIS.Control[nAxis].AxisState           := ADR(GVL_AXIS.State);         // state + result of command

  GVL_AXIS.Control[nAxis].Axes                REF=   GVL_AXIS.AxisRef;        // All for one; coupling requires access across all axes

  GVL_AXIS.Control[nAxis].AxisInfo            := ADR(GVL_AXIS.Info);          // axis information: act/set values and bits from axis
  GVL_AXIS.Control[nAxis].AxisData            := ADR(GVL_AXIS.Data);          // position and dynamic constraints for movement
  GVL_AXIS.Control[nAxis].AxisGearInParameter := ADR(GVL_AXIS.GearInParameter);

  GVL_AXIS.Control[nAxis].WriteNcParameter    := ADR(GVL_AXIS.NcParameterWrt);
  GVL_AXIS.Control[nAxis].ReadNcParameter     := ADR(GVL_AXIS.NcParameterRd);

  GVL_AXIS.Control[nAxis].HomingParameter     := ADR(GVL_AXIS.HomeParameter);
  GVL_AXIS.Control[nAxis].MotionOptions       := ADR(GVL_AXIS.MotionOptions);

  GVL_AXIS.ItfMcAxis[nAxis]                   := GVL_AXIS.Control[nAxis]; 
END_FOR
//-----------------------------------------------------------------------------------------------------------------
// assign dataflow/
//-----------------------------------------------------------------------------------------------------------------
//-----------------------------------------------------------------------------------------------------------------
// /INIT
//-----------------------------------------------------------------------------------------------------------------
IF NOT bInit
THEN
  CASE eInit
  OF
    E_PROGRESS.INVALID,
    E_PROGRESS.DONE:
      FOR nAxis := 1 TO MAX_AXIS
      DO
        GVL_AXIS.Control[nAxis].MessageLevel  := GVL_MSG.MessageLevel;
      END_FOR 
      nAxisInit                               := 1;
      eInit                                   := E_PROGRESS.INIT;


    E_PROGRESS.INIT:
      stMsg.eType                             := E_MessageType.eMessageVerbose;
      stMsg.eDevice                           := e_Device.General;
      stMsg.eSubdevice                        := e_SubDevice.AxisStartUp;
      stMsg.iErrorNumber                      := nAxisInit;

      stMsg.sText                             := concat('MAIN.eInit: ', TO_STRING(eInit));
      f_MessageSet(stMsg);

      GVL_AXIS.Ctrl[nAxisInit].eCtrl          := E_AXIS_CTRL.AXIS_NULL;
      eInit                                   := E_PROGRESS.BUSY;


    E_PROGRESS.BUSY:
      GVL_AXIS.Ctrl[nAxisInit].eCtrl          := E_AXIS_CTRL.AXIS_INIT;

      IF    (GVL_AXIS.State[nAxisInit].eState = E_AXIS_STATE.AXIS_INIT + E_PROGRESS.ERROR)
      THEN
        eInit                                 := E_PROGRESS.ERROR;

        stMsg.eType                           := E_MessageType.eMessageError;
        stMsg.eDevice                         := e_Device.General;
        stMsg.eSubdevice                      := e_SubDevice.AxisStartUp;
        stMsg.iErrorNumber                    := GVL_AXIS.Control[nAxisInit].ErrorId;

        stMsg.sText                           := concat('MAIN.eInit ERROR at Index: ', TO_STRING(nAxisInit));
        f_MessageSet(stMsg);

      ELSIF (GVL_AXIS.State[nAxisInit].eState = E_AXIS_STATE.AXIS_INIT + E_PROGRESS.DONE)
      THEN
        eInit                                 := E_PROGRESS.READY;
      END_IF


    E_PROGRESS.READY:
      IF NOT (nAxisInit > PLC_CONSTANT.MAX_AXIS-1)
      THEN
        nAxisInit                             := nAxisInit + 1;
        eInit                                 := E_PROGRESS.INIT;

      ELSE
        bInit                                 := TRUE;
        eInit                                 := E_PROGRESS.DONE;

        stMsg.eType                           := E_MessageType.eMessageInfo;
        stMsg.eDevice                         := e_Device.General;
        stMsg.eSubdevice                      := e_SubDevice.AxisStartUp;
        stMsg.iErrorNumber                    := MAX_AXIS;

        stMsg.sText                           := concat('MAIN.eInit: ', TO_STRING(eInit));
        f_MessageSet(stMsg);
      END_IF
  END_CASE
END_IF
//-----------------------------------------------------------------------------------------------------------------
// INIT
//-----------------------------------------------------------------------------------------------------------------
//-----------------------------------------------------------------------------------------------------------------
// /cyclic
//-----------------------------------------------------------------------------------------------------------------
IF (eInit <> E_PROGRESS.ERROR)
THEN
  FOR nAxis := 1 TO PLC_CONSTANT.MAX_AXIS
  DO
      GVL_AXIS.Control[nAxis]();
  END_FOR
END_IF
//-----------------------------------------------------------------------------------------------------------------
// cyclic/
//-----------------------------------------------------------------------------------------------------------------


//-----------------------------------------------------------------------------------------------------------------
// /logging
//-----------------------------------------------------------------------------------------------------------------
tonWriteLog(IN:= TRUE, PT := tWriteLog);

IF (tonWriteLog.Q)
THEN
  MessageData.bWriteFile      := TRUE;
  tonWriteLog(IN:= FALSE);
END_IF

//-----------------------------------------------------------------------------------------------------------------
// write message list to file
//-----------------------------------------------------------------------------------------------------------------
MessageData(pList			        := ADR(GVL_MSG.Messages),
			      pLocalTime        := ADR(GVL_MSG.dtLocalTime), 
			      bBusy=> );

// clear write trigger
IF MessageData.bWriteFile AND
   MessageData.bBusy
THEN
  MessageData.bWriteFile      := FALSE;
END_IF
//-----------------------------------------------------------------------------------------------------------------
// logging/
//-----------------------------------------------------------------------------------------------------------------

END_PROGRAM

// ---- _MSG/f_MessageSet.TcPOU
FUNCTION f_MessageSet : BOOL
VAR_INPUT
  stMessage   : ST_Message;
END_VAR
VAR
  _uiIndex   : uINT;
END_VAR

stMessage.tTime                     := GVL_MSG.sLocalTime;

IF (stMessage.eType = eMessageVerbose)
THEN
  IF NOT (GVL_MSG.MessageLevel = eMessageVerbose)
  THEN
    RETURN;
  END_IF
END_IF

IF (stMessage.eType = eMessageInfo)
THEN
  IF NOT (GVL_MSG.MessageLevel < eMessageError)
  THEN
    RETURN;
  END_IF
END_IF


FOR _uiIndex := 1 TO GVL_MSG.MAX_MESSAGE
DO
  IF (GVL_MSG.Messages[_uiIndex].eType = e_MessageType.eMessageEmpty)
  THEN
    GVL_MSG.Messages[_uiIndex]      := stMessage;
    GVL_MSG.MessageIndex            := _uiIndex;
    EXIT;
  END_IF
END_FOR

IF (stMessage.eType = E_MessageType.eMessageError)
THEN
  // in case of error: increment counter
  GVL_MSG.MessageError := GVL_MSG.MessageError + 1;
END_IF

END_FUNCTION

// ---- _MSG/MessageData.TcPOU
PROGRAM MessageData
VAR_INPUT
  bActivate     : BOOL;   // activates cyclic copy of message list to visualization; switched on in T_MESSAGE_LIST visu
	bPowerFail		: BOOL;   // UPS switch
	bWriteFile		: BOOL;   // manual write of list
	bReset				: BOOL;
	pList					: POINTER TO ARRAY[1..PLC_CONSTANT.MAX_MESSAGE] OF ST_Message; // attach your list here
	pLocalTime		: POINTER TO DT; 
END_VAR
VAR_OUTPUT
	bBusy					: BOOL;
  bDone         : BOOL;
	VisuList		  : ARRAY[1..PLC_CONSTANT.MAX_MESSAGE] OF ST_Message;
END_VAR
VAR
	eState 				: E_MESSAGE_STATE;

	rtrigReset		: Tc2_Standard.R_TRIG;
	aWriteList		: ARRAY[1..PLC_CONSTANT.MAX_MESSAGE] OF ST_Message;
	sWriteData		: STRING(32767);
	sNewLine			: STRING := '$N';
	sTab					: STRING := '$T';
	iCount, 
	iStart, 
	iEnd					: INT;

	fbCreateDir		: Tc2_System.FB_CreateDir;
	sTmp          : STRING(256);
	sFilename			: STRING(256);
	sFolderDate		: STRING;
	bFileCreated	: BOOL;

	fbFileOpen		  : Tc2_System.FB_FileOpen;
	fbFileWrite		  : Tc2_System.FB_FileWrite;
	fbFileClose		  : Tc2_System.FB_FileClose;

  ivis          : INT;

  bBusyWrite,
  bErrorWrite   : BOOL;
  nErrorWrite   : UDINT;
  nStateWrite   : UINT;
END_VAR

//-----------------------------------------------------------------------------
// check pointers
//-----------------------------------------------------------------------------
IF NOT (pList <> 0) OR
   NOT (pLocalTime <> 0)
THEN
  eState                      := MSG_INVALID_POINTERS;
  RETURN;
END_IF
//-----------------------------------------------------------------------------
// check date
// new message file for a new day
//-----------------------------------------------------------------------------
IF (FolderDate(pLocalTime) <> sFolderDate)
THEN
  bFileCreated                := FALSE;
END_IF
//-----------------------------------------------------------------------------
//----------------------------------------------------------------------------- 
rtrigReset(CLK:= bReset);
IF rtrigReset.Q
THEN
  bReset                      := FALSE;
  eState                      := MSG_NULL;
END_IF
//-----------------------------------------------------------------------------
//-----------------------------------------------------------------------------
CASE eState OF
  MSG_NULL:
    bBusy                     := 
    bDone                     := FALSE;
    
    IF (bWriteFile) OR
       (bPowerFail) OR 
       (GVL_MSG.MessageIndex > PLC_CONSTANT.MAX_MESSAGE-1)
    THEN
      eState                  := MSG_INIT;
    END_IF
END_CASE
//-----------------------------------------------------------------------------
CASE eState OF
  MSG_INIT:
    WriteData(FALSE);

    // clear intern list
    memset(ADR(aWriteList),     0, SIZEOF(aWriteList));

    // copy from attached list to local
    memcpy(ADR(aWriteList), pList, SIZEOF(aWriteList));

    // clear attached list
    memset(pList, 0, SIZEOF(aWriteList));

    bBusy                     := TRUE;
    iStart 	                  := 1;
    iEnd 		                  := SEL((GVL_MSG.MessageIndex > PLC_CONSTANT.MAX_MESSAGE-1),
                                      GVL_MSG.MessageIndex,
                                      PLC_CONSTANT.MAX_MESSAGE);
    GVL_MSG.MessageIndex      := 1;

    IF NOT bFileCreated
    THEN
      IF (GVL_MSG.MessageError > 0) OR
         (GVL_MSG.EnableLogging)
      THEN
        // folder and filename have to be created
        eState                := MSG_ROOT;
      ELSE
        eState                := MSG_WRITE_FILE_DONE; 
      END_IF
    ELSE
      // folder and file already exist
      eState                  := MSG_LINE_START;
    END_IF
END_CASE
//-----------------------------------------------------------------------------
CASE eState OF
  MSG_ROOT:
    eState                    := MSG_ROOT_CREATE;
    fbCreateDir.sPathName     := left(PLC_CONSTANT.LOG_DIR,len(PLC_CONSTANT.LOG_DIR)-1);
    fbCreateDir(
            bExecute	        := FALSE);
  
  MSG_ROOT_CREATE:
    (* create root folder *)
    fbCreateDir(
            bExecute	        := TRUE);
    IF fbCreateDir.bBusy
    THEN
      eState                  := MSG_ROOT_CREATE_BUSY;
    END_IF
  
  MSG_ROOT_CREATE_BUSY:
    fbCreateDir(
            bExecute	        := TRUE);
    IF NOT fbCreateDir.bBusy
    THEN
      eState                  := MSG_FOLDER;
    END_IF
  
  MSG_FOLDER:
    eState                    := MSG_FOLDER_CREATE;
    sFolderDate               := FolderDate(pLocalTime);
    fbCreateDir.sPathName     := concat(PLC_CONSTANT.LOG_DIR, sFolderDate);
    fbCreateDir(
            bExecute	        := FALSE);

  MSG_FOLDER_CREATE:
    (* create active folder *)
    fbCreateDir(
            bExecute	        := TRUE);
    IF fbCreateDir.bBusy
    THEN
      eState                  := MSG_FOLDER_CREATE_BUSY;
    END_IF
  
  MSG_FOLDER_CREATE_BUSY:
    fbCreateDir(
            bExecute	        := TRUE);
    IF NOT fbCreateDir.bBusy
    THEN
      eState                  := MSG_FILE_CREATE_DONE;
      fbCreateDir(
              bExecute	      := FALSE);
    END_IF
END_CASE
//-----------------------------------------------------------------------------
CASE eState OF
  MSG_FILE_CREATE_DONE:
    eState                    := MSG_LINE_START;
    bFileCreated              := TRUE;
    // build complete file path
    sTmp                      := concat(concat(PLC_CONSTANT.LOG_FILE, sFolderDate),'.txt');
    sTmp                      := concat('\', sTmp);
    sFilename                 := concat(fbCreateDir.sPathName, sTmp);
END_CASE
//-----------------------------------------------------------------------------
CASE eState OF
  MSG_LINE_START:
    GVL_MSG.MessageError      := 0;
    eState                    := MSG_LINE_BUILD;
    iCount                    := iStart;
    memset(ADR(sWriteData),0,SIZEOF(sWriteData));
END_CASE
//-----------------------------------------------------------------------------
CASE eState OF
  MSG_LINE_BUILD:
    eState                    := MSG_LINE_CHECK;
    IF (aWriteList[iCount].eType > E_MessageType.eMessageEmpty)
    THEN
      IF (aWriteList[iCount].eType > E_MessageType.eMessageInfo) OR
         (GVL_MSG.EnableLogging)
      THEN
        sTmp                  := TO_STRING(aWriteList[iCount].eType);
        sTmp                  := Tc2_Standard.CONCAT(sTmp, sTab);
        sTmp                  := Tc2_Standard.CONCAT(sTmp, aWriteList[iCount].tTime);
        sTmp                  := Tc2_Standard.CONCAT(sTmp, sTab);
        sTmp                  := Tc2_Standard.CONCAT(sTmp, Device_To_String(aWriteList[iCount].eDevice));
        sTmp                  := Tc2_Standard.CONCAT(sTmp, sTab);
        sTmp                  := Tc2_Standard.CONCAT(sTmp, TO_STRING(aWriteList[iCount].eSubdevice));
        sTmp                  := Tc2_Standard.CONCAT(sTmp, sTab);
        sTmp                  := Tc2_Standard.CONCAT(sTmp, TO_STRING(aWriteList[iCount].iErrorNumber));
        sTmp                  := Tc2_Standard.CONCAT(sTmp, sTab);
        sTmp                  := Tc2_Standard.CONCAT(sTmp, aWriteList[iCount].sText);
        sTmp                  := Tc2_Standard.CONCAT(sTmp, sNewLine);
        Builder(ADR(sTmp), ADR(sWriteData), StringLen(ADR(sTmp)));
      END_IF
    END_IF
    iCount                    := iCount + 1;
END_CASE
//-----------------------------------------------------------------------------
CASE eState OF
  MSG_LINE_CHECK:
  IF NOT (iCount > iEnd)
  THEN
    eState                    := MSG_LINE_BUILD;
  ELSE
    IF (StringLen(ADR(sWriteData)) > 1)
    THEN
      eState                  := MSG_WRITE_FILE_BUSY;
    ELSE
      eState                  := MSG_WRITE_FILE_DONE;
    END_IF
  END_IF
  
  MSG_WRITE_FILE_BUSY:
  IF WriteData(TRUE)
  THEN
    eState                    := MSG_WRITE_FILE_END;
  END_IF
  
  MSG_WRITE_FILE_END:
  WriteData(FALSE);
  eState                      := MSG_WRITE_FILE_DONE;
  
  MSG_WRITE_FILE_DONE:
  bDone                       := TRUE;
  IF NOT (bWriteFile)
  THEN
    eState                    := MSG_NULL;
  END_IF
END_CASE
//-----------------------------------------------------------------------------
//-----------------------------------------------------------------------------
// visu message list
//-----------------------------------------------------------------------------
memset(ADR(VisuList),0,SIZEOF(VisuList));

IF (bActivate)
THEN
  // copy message list to visu message list
  FOR ivis := 1 TO GVL_MSG.MessageIndex
  DO
    VisuList[ivis]            := pList^[ivis];
  END_FOR
END_IF
//-----------------------------------------------------------------------------

METHOD Builder : BOOL // string concat for length > 255
VAR_INPUT
  pInString   : POINTER TO STRING;
  pOutString  : POINTER TO STRING(32767);
  Length      : UINT;
END_VAR
VAR
  Counter     : DINT;
  pInWork     : POINTER TO BYTE;
  pOutWork    : POINTER TO BYTE;
END_VAR
pOutWork := pOutString;
pInWork := pInString;
Counter := 0;

(*check termination*)
WHILE (pOutWork^ <> 0) AND
      (Counter < 32767)
DO
  Counter := Counter + 1;
  pOutWork := pOutWork + 1;
END_WHILE

(* append only if data fits into output *)
IF (Counter + Length < 32767)
THEN

  (* append data *)
  FOR Counter := 1 TO Length
  DO
    pOutWork^ := pInWork^;
    pOutWork := pOutWork + 1;
    pInWork := pInWork + 1;
  END_FOR

  (* terminate *)
  pOutWork := pOutWork + 1;
  pOutWork^ := 0;
END_IF
END_METHOD

METHOD Device_to_String : string
VAR_INPUT
  eMsgDevice    : e_Device;
END_VAR
VAR
  // first NC Axis, all other Axis are incremented
  nmodAxis            : DINT := 1000;

  // first NCI channel control instance
  nmodNciChannelCtrl  : DINT := 2000;

  // NCI channel
  nmodNciChannel      : DINT := 3000;

  // CAMMING
  nmodCamming         : DINT := 6000;

  // message function blocks
  nmodData            : DINT := 10000;

  sId                 : STRING := '_ID_';
  nId                 : DINT;
END_VAR

IF (eMsgDevice <= nmodAxis)
THEN
  // general case with no added indices
  Device_to_String := TO_STRING(eMsgDevice);
ELSE

  IF (eMsgDevice > nModData)
  THEN
    nId := eMsgDevice MOD nmodData;
    sId := concat(sId, TO_STRING(nId));
 
    Device_to_String := concat(TO_STRING(e_device.Data), sId);

  ELSIF (eMsgDevice > nmodCamming)
  THEN
    nId := eMsgDevice MOD nmodCamming;
    sId := concat(sId, TO_STRING(nId));
    sId := concat('_AXIS', sId);
 
    Device_to_String := concat(TO_STRING(e_device.Camming), sId);

  ELSIF (eMsgDevice > nmodNciChannel)
  THEN
    nId := eMsgDevice MOD nmodNciChannel;
    sId := concat(sId, TO_STRING(nId));
 
    Device_to_String := concat(TO_STRING(e_device.NciChannel), sId);

  ELSIF (eMsgDevice > nmodNciChannelCtrl)
  THEN
    nId := eMsgDevice MOD nmodNciChannelCtrl;
    sId := concat(sId, TO_STRING(nId));
 
    Device_to_String := concat(TO_STRING(e_device.NciChannelCtrl), sId);

  ELSIF (eMsgDevice > nmodAxis)
  THEN
    nId := eMsgDevice MOD nmodAxis;
    sId := concat(sId, TO_STRING(nId));
 
    Device_to_String := concat(TO_STRING(e_device.Axis), sId);
  ELSE
    Device_to_String := TO_STRING(eMsgDevice);
  END_IF
END_IF
END_METHOD

METHOD FolderDate : STRING
VAR_INPUT
	pLocalTime		: POINTER TO DT;
END_VAR
VAR
	sTmp					: STRING;
END_VAR
IF NOT (pLocalTime <> 0)
THEN
	FolderDate := 'NULL';
	RETURN;
END_IF

sTmp := DT_TO_STRING(pLocalTime^);

// cut off #dt literal
sTmp := right(sTmp, len(sTmp)-3);

sTmp := replace(sTmp, '_', 1, 5);
sTmp := replace(sTmp, '_', 1, 8);

sTmp := left(sTmp,10);	// year_month_day

FolderDate := sTmp;
END_METHOD

METHOD StringLen : UINT // 	string length for len > 255
VAR_INPUT
  pInString		: POINTER TO STRING(32767);
END_VAR
VAR
	Counter			: UINT;
	pInWork			: POINTER TO BYTE;
END_VAR
pInWork := pInString;
Counter := 0;

WHILE (pInWork^ <> 0) AND
			(Counter < 32767)
DO
	Counter := Counter + 1;
	pInWork := pInWork + 1;
END_WHILE

StringLen := Counter;
END_METHOD

METHOD WriteData  : BOOL
VAR_INPUT
  bExecute        : BOOL;
END_VAR
VAR
END_VAR

IF NOT bExecute
THEN
  bBusyWrite                := FALSE;
	nStateWrite               := 0;
END_IF

CASE nStateWrite OF

	0:
		fbFileOpen.bExecute		  := FALSE;
		fbFileWrite.bExecute	  := FALSE;
		fbFileClose.bExecute	  := FALSE;

		IF bExecute
		THEN
			bBusyWrite            := TRUE;
			nStateWrite           := 10;
		END_IF

	10:
		fbFileOpen.bExecute     := TRUE;
		IF fbFileOpen.bBusy
		THEN
			nStateWrite           := 20;
		END_IF

	20:
		IF NOT fbFileOpen.bBusy
		THEN
			fbFileOpen.bExecute   := FALSE;
			fbFileWrite.bExecute  := TRUE;
			nStateWrite           := 30;
		END_IF

	30:
		IF fbFileWrite.bBusy
		THEN
			nStateWrite           := 40;
		END_IF

	40:
		IF NOT fbFileWrite.bBusy
		THEN
			fbFileWrite.bExecute  := FALSE;
			fbFileClose.bExecute  := TRUE;
			nStateWrite           := 50;
		END_IF

	50:
		IF fbFileClose.bBusy
		THEN
			nStateWrite           := 60;
		END_IF

	60:
		IF NOT fbFileClose.bBusy
		THEN
			fbFileClose.bExecute  := FALSE;
			nStateWrite 		      := 100;
		END_IF
	
	100:
    WriteData               := TRUE;
END_CASE


fbFileOpen(
	sNetId:= , 
	sPathName:= sFileName, 
	nMode:= FOPEN_MODEAPPEND, 
	ePath:= PATH_GENERIC, 
	bExecute:= , 
	tTimeout:= T#10S, 
	bBusy=> , 
	bError=> , 
	nErrId=> , 
	hFile=> );

fbFileWrite(
	sNetId:= , 
	hFile:= fbFileOpen.hFile, 
	pWriteBuff:= ADR(sWriteData), 
	cbWriteLen:= StringLen(ADR(sWriteData)), 
	bExecute:= , 
	tTimeout:= T#10S, 
	bBusy=> , 
	bError=> , 
	nErrId=> nErrorWrite, 
	cbWrite=> );

fbFileClose(
	sNetId:= , 
	hFile:= fbFileOpen.hFile, 
	bExecute:= , 
	tTimeout:= T#10S, 
	bBusy=> , 
	bError=> , 
	nErrId=> );

bErrorWrite := fbFileOpen.bError OR fbFileWrite.bError;
END_METHOD

END_PROGRAM

// ---- NCI.TcPOU
PROGRAM NCI
VAR
  bInit                     : BOOL;
  eInit                     : E_PROGRESS;

  nChn,
  nChnInit,
  nAxis,
  nAxisInit                 : UINT;

  stMsg                     : ST_Message;

END_VAR

//-----------------------------------------------------------------------------------------------------------------
// check if compiler define is present [PLC_STATE_DRIVE/CompilerDefines/Manual: NCI]
// see PLC_CONSTANT for conditional pragma
//-----------------------------------------------------------------------------------------------------------------
IF NOT PLC_CONSTANT.NCI_ACTIVE THEN eInit   := E_PROGRESS.NOT_EXIST; RETURN; END_IF
//-----------------------------------------------------------------------------------------------------------------
//-----------------------------------------------------------------------------------------------------------------
//-----------------------------------------------------------------------------------------------------------------
//-----------------------------------------------------------------------------------------------------------------
// /assign dataflow
//-----------------------------------------------------------------------------------------------------------------
FOR nChn := 1 TO MAX_NCI_CH
DO
  GVL_NCI.fbNciCtrl[nChn].ItfChannel.MessageLevel     := GVL_MSG.MessageLevelNciChn[nChn];

  // NCI axis configuration --> NC AxisId used
  GVL_NCI.fbNciCtrl[nChn].ItfChannel.CfgAxes          := ADR(GVL_NCI.stAxisConfig[nChn]);

  // R Parameter properties
  GVL_NCI.fbNciCtrl[nChn].ItfChannel.R_ParameterRead  := ADR(GVL_NCI.R_ParameterRead[nChn]);
  GVL_NCI.fbNciCtrl[nChn].ItfChannel.R_ParameterWrite := ADR(GVL_NCI.R_ParameterWrite[nChn]);

  // ProgName for channel
  GVL_NCI.fbNciCtrl[nChn].ItfChannel.Prog             := GVL_NCI.sProgName[nChn];

  // check REAL value to avoid exception
  IF NOT IsFinite(F_Real(GVL_NCI.stChannelCtrl[nChn].rOverride))
  THEN
    GVL_NCI.fbNciCtrl[nChn].ItfChannel.Override       := 0.0;
  ELSE
    GVL_NCI.fbNciCtrl[nChn].ItfChannel.Override       := GVL_NCI.stChannelCtrl[nChn].rOverride;
  END_IF

  // command and state structure assignement
  GVL_NCI.fbNciCtrl[nChn].ChnCtrl                     := ADR(GVL_NCI.stChannelCtrl[nChn]);
  GVL_NCI.fbNciCtrl[nChn].ChnState                    := ADR(GVL_NCI.stChannelState[nChn]);
END_FOR
//-----------------------------------------------------------------------------------------------------------------
// assign dataflow/
//-----------------------------------------------------------------------------------------------------------------
//-----------------------------------------------------------------------------------------------------------------
// /INIT
//-----------------------------------------------------------------------------------------------------------------
IF NOT bInit
THEN
  CASE eInit
  OF
    E_PROGRESS.INVALID,
    E_PROGRESS.DONE:
      FOR nChn := 1 TO MAX_NCI_CH
      DO
        GVL_MSG.MessageLevelNciChn[nChn]          := GVL_MSG.MessageLevel;
      END_FOR 
      nChnInit                                    := 1;
      eInit                                       := E_PROGRESS.INIT;


    E_PROGRESS.INIT:
      stMsg.eType                                 := E_MessageType.eMessageVerbose;
      stMsg.eDevice                               := e_Device.NciChannelCtrl;
      stMsg.eSubdevice                            := e_SubDevice.NciStartUp;
      stMsg.iErrorNumber                          := nChnInit;

      stMsg.sText                                 := concat('NCI.eInit: ', TO_STRING(eInit));
      f_MessageSet(stMsg);

      GVL_NCI.stChannelCtrl[nChnInit].eCmd        := E_NCI_CTRL.NULL;
      eInit                                       := E_PROGRESS.BUSY;


    E_PROGRESS.BUSY:
      GVL_NCI.stChannelCtrl[nChnInit].eCmd        := E_NCI_CTRL.INIT;

      IF (GVL_NCI.stChannelState[nChnInit].eState = E_NCI_STATE.INIT + E_PROGRESS.ERROR)
      THEN
        eInit                                     := E_PROGRESS.ERROR;

        stMsg.eType                               := E_MessageType.eMessageError;
        stMsg.eDevice                             := e_Device.NciChannelCtrl;
        stMsg.eSubdevice                          := e_SubDevice.NciStartUp;
        stMsg.iErrorNumber                        := nChnInit;

        stMsg.sText                               := concat('NCI.eInit ERROR at Index: ', TO_STRING(nChnInit));
        f_MessageSet(stMsg);

      ELSIF (GVL_NCI.stChannelState[nChnInit].eState = E_NCI_STATE.INIT + E_PROGRESS.DONE)
      THEN
        eInit                                     := E_PROGRESS.READY;
      END_IF


    E_PROGRESS.READY:
      IF (nChnInit > PLC_CONSTANT.MAX_NCI_CH-1)
      THEN
        bInit                                     := TRUE;
        eInit                                     := E_PROGRESS.DONE;

        stMsg.eType                               := E_MessageType.eMessageInfo;
        stMsg.eDevice                             := e_Device.NciChannelCtrl;
        stMsg.eSubdevice                          := e_SubDevice.NciStartUp;
        stMsg.iErrorNumber                        := MAX_NCI_CH;

        stMsg.sText                               := concat('NCI.eInit: ', TO_STRING(eInit));
        f_MessageSet(stMsg);

      ELSE
        nChnInit                                  := nChnInit + 1;
        eInit                                     := E_PROGRESS.INIT;
      END_IF
  END_CASE
END_IF
//-----------------------------------------------------------------------------------------------------------------
// INIT
//-----------------------------------------------------------------------------------------------------------------
//-----------------------------------------------------------------------------------------------------------------
//-----------------------------------------------------------------------------------------------------------------
// /CYCLE
//-----------------------------------------------------------------------------------------------------------------
FOR nChn := 1 TO MAX_NCI_CH
DO
  // call nci channel controller
  GVL_NCI.fbNciCtrl[nChn].Cycle();

  GVL_NCI.sProgNameActive[nChn]             := GVL_NCI.fbNciCtrl[nChn].ItfChannel.GetLoadedProg();
  GVL_NCI.fbNciCtrl[nChn].M_FunctionScope   := ADR(GVL_NCI.M_FunctionCyclic[nChn]);
END_FOR
//-----------------------------------------------------------------------------------------------------------------
// CYCLE/
//-----------------------------------------------------------------------------------------------------------------
//-----------------------------------------------------------------------------------------------------------------

END_PROGRAM

// ---- CAM.TcPOU
PROGRAM CAM
VAR
  bInit                     : BOOL;
  eInit                     : E_PROGRESS;

  nAxis,
  nAxisInit                 : UINT;

  stMsg                     : ST_Message;
END_VAR

//-----------------------------------------------------------------------------------------------------------------
// check if compiler define is present [PLC_STATE_DRIVE/CompilerDefines/Manual: CAM]
// see PLC_CONSTANT for conditional pragma
//-----------------------------------------------------------------------------------------------------------------
IF NOT PLC_CONSTANT.CAM_ACTIVE THEN eInit := E_PROGRESS.NOT_EXIST; RETURN; END_IF
//-----------------------------------------------------------------------------------------------------------------
//-----------------------------------------------------------------------------------------------------------------
//-----------------------------------------------------------------------------------------------------------------
//-----------------------------------------------------------------------------------------------------------------
// /assign dataflow
//-----------------------------------------------------------------------------------------------------------------
FOR nAxis := 1 TO PLC_CONSTANT.MAX_AXIS
DO
  GVL_CAM.Control[nAxis].ItfMcAxes                := GVL_AXIS.ItfMcAxis;
  GVL_CAM.Control[nAxis].MessageLevel             := GVL_MSG.MessageLevelAxisCam[nAxis];

  GVL_CAM.Control[nAxis].AxisIndex                := nAxis;

  GVL_CAM.Control[nAxis].AxisCtrl                 := ADR(GVL_CAM.Ctrl);          // command
  GVL_CAM.Control[nAxis].AxisState                := ADR(GVL_CAM.State);         // state + result of command

  GVL_CAM.Control[nAxis].Axes                     REF=   GVL_AXIS.AxisRef;        // All for one; coupling requires access across all axes

  GVL_CAM.Control[nAxis].AxisInfo                 := ADR(GVL_CAM.Info);
  GVL_CAM.Control[nAxis].AxisData                 := ADR(GVL_CAM.Data);

  GVL_CAM.Control[nAxis].MotionFunction           := ADR(GVL_CAM.MotionFunction);
  GVL_CAM.Control[nAxis].MotionFunctionPoint      := ADR(GVL_CAM.MotionFunctionPoint);
END_FOR
//-----------------------------------------------------------------------------------------------------------------
// assign dataflow/
//-----------------------------------------------------------------------------------------------------------------
//-----------------------------------------------------------------------------------------------------------------
// /INIT
//-----------------------------------------------------------------------------------------------------------------
IF NOT bInit
THEN
  CASE eInit
  OF
    E_PROGRESS.INVALID,
    E_PROGRESS.DONE:
      FOR nAxis := 1 TO MAX_AXIS
      DO
        GVL_CAM.Control[nAxis].MessageLevel       := GVL_MSG.MessageLevel;
      END_FOR 
      nAxisInit                                   := 1;
      eInit                                       := E_PROGRESS.INIT;


    E_PROGRESS.INIT:
      stMsg.eType                                 := E_MessageType.eMessageVerbose;
      stMsg.eDevice                               := e_Device.Camming;
      stMsg.eSubdevice                            := e_SubDevice.CamStartUp;
      stMsg.iErrorNumber                          := nAxisInit;

      stMsg.sText                                 := concat('CAM.eInit: ', TO_STRING(eInit));

      f_MessageSet(stMsg);

      GVL_CAM.Ctrl[nAxisInit].eCtrl               := E_AXIS_CTRL.AXIS_NULL;
      eInit                                       := E_PROGRESS.BUSY;


    E_PROGRESS.BUSY:
      GVL_CAM.Ctrl[nAxisInit].eCtrl               := E_AXIS_CTRL.AXIS_INIT;

      IF (GVL_CAM.State[nAxisInit].eState = E_AXIS_STATE.AXIS_INIT + E_PROGRESS.ERROR)
      THEN
        eInit                                     := E_PROGRESS.ERROR;

        stMsg.eType                               := E_MessageType.eMessageError;
        stMsg.eDevice                             := e_Device.Camming;
        stMsg.eSubdevice                          := e_SubDevice.CamStartUp;
        stMsg.iErrorNumber                        := nAxisInit;

        stMsg.sText                               := concat('CAM.eInit ERROR at Index: ', TO_STRING(nAxisInit));
        f_MessageSet(stMsg);

      ELSIF (GVL_CAM.State[nAxisInit].eState = E_AXIS_STATE.AXIS_INIT + E_PROGRESS.DONE)
      THEN
        eInit                                     := E_PROGRESS.READY;
      END_IF


    E_PROGRESS.READY:
      IF (nAxisInit > PLC_CONSTANT.MAX_AXIS-1)
      THEN
        bInit                                     := TRUE;
        eInit                                     := E_PROGRESS.DONE;

        stMsg.eType                               := E_MessageType.eMessageInfo;
        stMsg.eDevice                             := e_Device.Camming;
        stMsg.eSubdevice                          := e_SubDevice.CamStartUp;
        stMsg.iErrorNumber                        := MAX_AXIS;

        stMsg.sText                               := concat('CAM.eInit: ', TO_STRING(eInit));
        f_MessageSet(stMsg);

      ELSE
        nAxisInit                                 := nAxisInit + 1;
        eInit                                     := E_PROGRESS.INIT;
      END_IF
  END_CASE
END_IF
//-----------------------------------------------------------------------------------------------------------------
// INIT
//-----------------------------------------------------------------------------------------------------------------
//-----------------------------------------------------------------------------------------------------------------
// /cyclic
//-----------------------------------------------------------------------------------------------------------------
IF (eInit <> E_PROGRESS.ERROR)
THEN
  FOR nAxis := 1 TO PLC_CONSTANT.MAX_AXIS
  DO
      GVL_CAM.Control[nAxis].Cycle();
  END_FOR
END_IF
//-----------------------------------------------------------------------------------------------------------------
// cyclic/
//-----------------------------------------------------------------------------------------------------------------

END_PROGRAM

// ---- MAPPING/MAPPING_out.TcPOU
PROGRAM MAPPING_out
VAR CONSTANT
{IF defined (AXIS_MAP)}
  {info 'MAPPING_out - ACTIVE'}
  bBypassMapping    : BOOL  := FALSE;
{ELSE}
  bBypassMapping    : BOOL  := TRUE;
{END_IF}
END_VAR
VAR
{IF defined (AXIS_MAP)}
  AxisState         : U_AXIS_STATE;
  AxisInfo          : U_AXIS_INFO;
  AxisParameterRd   : U_AXIS_NC_PARAMETER_RD;
{ELSE}
  AxisState         : BYTE;
  AxisInfo          : BYTE;
  AxisParameterRd   : BYTE;
{END_IF}
END_VAR

IF bBypassMapping THEN RETURN; END_IF

memcpy(ADR(AxisState),         ADR(GVL_AXIS.State),             SIZEOF(GVL_AXIS.State));
memcpy(ADR(AxisInfo),          ADR(GVL_AXIS.Info),              SIZEOF(GVL_AXIS.Info));
memcpy(ADR(AxisParameterRd),   ADR(GVL_AXIS.NcParameterRd),     SIZEOF(GVL_AXIS.NcParameterRd));

END_PROGRAM

// ---- NC_PTP/FB_McAxisCtrl.TcPOU
FUNCTION_BLOCK FB_McAxisCtrl EXTENDS FB_McAxis IMPLEMENTS I_McAxis
VAR
  _eCheck                   : E_CHECK_STATE;  // pointer check

  _eAxisCycle,                                // cyclic AXIS_REF() and MC_Power check
  _eInit                    : E_PROGRESS;     // axis startup and init, get encoder type, get axis name, get device name

  _nAxisIndex               : UINT;           // know thyself
  _rTargetWindow            : LREAL := 0.1;   // TODO: get that from NC

  // pointers to all; access required for coupling; access by index
  _Axes                     : REFERENCE TO ARRAY[1..PLC_CONSTANT.MAX_AXIS] OF AXIS_REF;

  _Ctrl                     : POINTER TO ARRAY[1..PLC_CONSTANT.MAX_AXIS] OF ST_AXIS_CTRL;    // contains command to be executed
  _State                    : POINTER TO ARRAY[1..PLC_CONSTANT.MAX_AXIS] OF ST_AXIS_STATE;   // mirrors command with added result

  _Info                     : POINTER TO ARRAY[1..PLC_CONSTANT.MAX_AXIS] OF ST_AXIS_INFO;    // axis state and position data to read from
  _Data                     : POINTER TO ARRAY[1..PLC_CONSTANT.MAX_AXIS] OF ST_MOVE_DATA;    // structure for cyclic interface

  _NcParameterWrt           : POINTER TO ARRAY[1..PLC_CONSTANT.MAX_AXIS] OF ST_NC_PARAMETER; // W struct for a single parameter
  _NcParameterRd            : POINTER TO ARRAY[1..PLC_CONSTANT.MAX_AXIS] OF ST_NC_PARAMETER; // R struct for a single parameter
  _HomeParameter            : POINTER TO ARRAY[1..PLC_CONSTANT.MAX_AXIS] OF ST_HOMING;       // homing parameter for each axis

  _GearInParameter          : POINTER TO ARRAY[1..PLC_CONSTANT.MAX_AXIS] OF ST_GEAR_IN;      // Master Indices, dyn constraints for simple GearIn

  _MotionOptions            : POINTER TO ARRAY[1..PLC_CONSTANT.MAX_AXIS] OF ST_MOTION_OPTIONS;


  // local copies of command
  _eCtrl,
  _eCtrlOld                       : E_AXIS_CTRL;

  // Last handled NC Axis parameter to write
  _eParameterNrWrite              : Tc2_MC2.MC_AxisParameter;
  _rParameterWrtValue             : LREAL;

  // Last handled NC Axis parameter to read
  _eParameterNrRead               : Tc2_MC2.MC_AxisParameter;
  _rParameterReadValue            : LREAL;

  // execution state
  _eResult                        : E_PROGRESS;   // result of execution state
  _eResultOld                     : E_PROGRESS;   // old result for detecting change
  _eState                         : E_AXIS_STATE; // execution state

  // calibration options with limit switches and simulation
  _bCalibrationCam                : BOOL;

  // mapping inputs
  _bLimitMin,
  _bLimitMax,
  _bCalibrationInput     AT %I*   : BOOL;


  // placeholder dummies in case count of Multimaster ases <> 4
  {attribute 'hide'}
  _MultiMasterDummyRef            : ARRAY[1..4] OF AXIS_REF;

  _fbGearOut                      : Tc2_MC2.MC_GearOut;
  _fbGearIn                       : Tc2_MC2.MC_GearIn;
  _fbGearInMultiMaster            : Tc2_MC2.MC_GearInMultiMaster;
END_VAR

IF NOT Check() THEN RETURN; END_IF
//-----------------------------------------------------------------------------
// check _HomeParameter for calibration input options
//-----------------------------------------------------------------------------
_bCalibrationCam                    := GetCalibrationCam();
CalibrationCam                      := ADR(_bCalibrationCam);
//-----------------------------------------------------------------------------
//-----------------------------------------------------------------------------
Override                            := _Data^[_nAxisIndex].rOverride;
//-----------------------------------------------------------------------------
//-----------------------------------------------------------------------------
// cyclic call to MC_Power and AXIS_REF()
//-----------------------------------------------------------------------------
_eAxisCycle                         := Cycle();
//-----------------------------------------------------------------------------
//-----------------------------------------------------------------------------
// get command from outside world
//-----------------------------------------------------------------------------
_eCtrl                              := _Ctrl^[_nAxisIndex].eCtrl;
//-----------------------------------------------------------------------------
//-----------------------------------------------------------------------------
//  OnChange react to command
//-----------------------------------------------------------------------------
IF (_eCtrl <> _eCtrlOld)
THEN
  // get busy
  _eState                           := Cmd(_eCtrl); // get execution state for command
  _eCtrlOld                         := _eCtrl;
  LogControl();
END_IF
//-----------------------------------------------------------------------------
//-----------------------------------------------------------------------------
// Check AxisInit
//-----------------------------------------------------------------------------
IF NOT (_eInit = E_PROGRESS.DONE)
THEN
  _Info^[_nAxisIndex].bReady        := FALSE;
ELSE
  _Info^[_nAxisIndex].bReady        := _AxisRef.Status.ControlLoopClosed AND
                                       (NOT _AxisRef.Status.Error)       AND 
                                       (NOT _AxisRef.Status.Moving);
END_IF
//-----------------------------------------------------------------------------
//-----------------------------------------------------------------------------
//  _eAxisCycle := Cycle() is called at the top; checks MC_Power.bError
//  MC_Power.bError requires e_AXIS_CTRL.AXIS_RESET in order to clear
//-----------------------------------------------------------------------------
CASE _eAxisCycle
OF
  E_PROGRESS.ERROR:
    _eResult                        := _eAxisCycle;
END_CASE
//-----------------------------------------------------------------------------
//-----------------------------------------------------------------------------
//  execution result
//-----------------------------------------------------------------------------
CASE _eResult
OF
  E_PROGRESS.INVALID:
    _State^[_nAxisIndex].eState     := TO_UINT(E_PROGRESS.ERROR);

  E_PROGRESS.ERROR:
    _Info^[_nAxisIndex].bReady      := FALSE;
    _Info^[_nAxisIndex].bError      := TRUE;
    _Info^[_nAxisIndex].nErrorId    := ErrorId;

    _State^[_nAxisIndex].eState     := _eState + E_PROGRESS.ERROR;

  E_PROGRESS.DONE:
    _State^[_nAxisIndex].eState     := _eState + E_PROGRESS.DONE;

ELSE
  //-----------------------------------------------------------------------------
  // execution state result to interface
  //-----------------------------------------------------------------------------
  _State^[_nAxisIndex].eState       := _eState + _eResult;

  //-----------------------------------------------------------------------------
  //-----------------------------------------------------------------------------
  //  execution state for command
  //-----------------------------------------------------------------------------
  CASE _eState
  OF
    E_AXIS_STATE.AXIS_INIT:
      //-------------------------------------------------------------------------
      // axis always requires one init from outside world at startup
      // _eInit has to be valid for other commands to be accepted in Cmd(_eCtrl)
      _eInit := _eResult            := AxisInit(TRUE);
  
    E_AXIS_STATE.AXIS_NO_INIT:
      //-------------------------------------------------------------------------
      // we are here because you sent a command before having done AXIS_INIT
      _eResult                      := E_PROGRESS.ERROR;
  
    E_AXIS_STATE.AXIS_DISABLE:
      _eResult                      := AxisDisable(TRUE);
  
    E_AXIS_STATE.AXIS_ENABLE:
      _eResult                      := AxisEnable(TRUE);
  
    E_AXIS_STATE.AXIS_IDLE:
      _eResult                      := AxisIdle(TRUE);
  
    E_AXIS_STATE.AXIS_HOME:
      _eResult                      := AxisHome(TRUE);
  
    E_AXIS_STATE.AXIS_MOVE_POS:
      _eResult                      := AxisMoveToPosition(TRUE, _Data^[_nAxisIndex]);
  
    E_AXIS_STATE.AXIS_MOVE_VELO:
      _eResult                      := AxisMoveVelocity(TRUE, _Data^[_nAxisIndex]);
  
    E_AXIS_STATE.AXIS_RESET:
      _eResult                      := AxisReset(TRUE);
  
    E_AXIS_STATE.AXIS_HALT:
      _eResult                      := AxisHalt(TRUE, _Data^[_nAxisIndex]);
  
    E_AXIS_STATE.AXIS_STOP:
      _eResult                      := AxisStop(TRUE, _Data^[_nAxisIndex]);
  
    E_AXIS_STATE.AXIS_MOVE_BUFFER:
      _eResult                      := AxisBufferPos(TRUE, _Data^[_nAxisIndex]);
  
    E_AXIS_STATE.AXIS_MOVE_BUFFER_VELO:
      _eResult                      := AxisBufferVelo(TRUE, _Data^[_nAxisIndex]);
  
    E_AXIS_STATE.AXIS_PARAMETER_READ:
      _eResult                      := AxisParameterRead(TRUE, _NcParameterRd^[_nAxisIndex].ParameterNumber);
  
    E_AXIS_STATE.AXIS_PARAMETER_WRITE:
      _eResult                      := AxisParameterWrite(TRUE, _NcParameterWrt^[_nAxisIndex].ParameterNumber);
  
    E_AXIS_STATE.AXIS_PARAMETER_WRITE_PERSISTENT:
      _eResult                      := AxisParameterWritePersistent(TRUE, _NcParameterWrt^[_nAxisIndex].ParameterNumber);
  
    E_AXIS_STATE.AXIS_GEAR_IN:
      _eResult                      := AxisGearIn(TRUE);
  
    E_AXIS_STATE.AXIS_GEAR_OUT:
      _eResult                      := AxisGearOut(TRUE);
  
    E_AXIS_STATE.AXIS_GEAR_IN_MULTIMASTER:
      _eResult                      := AxisGearInMultiMaster(TRUE);
  
  ELSE
    IF (_eCtrl > E_AXIS_CTRL.AXIS_NULL)
    THEN
      _eResult                      := E_PROGRESS.NOT_EXIST;
      _Info^[_nAxisIndex].bError    := TRUE;
    ELSE
      _eResult                      := E_PROGRESS.INVALID;
    END_IF
  END_CASE
END_CASE
//-----------------------------------------------------------------------------
//-----------------------------------------------------------------------------
//  OnChange of execution state result
//    - log result and clear error number on interface
//-----------------------------------------------------------------------------
IF (_eResult <> _eResultOld)
THEN
  LogResult();
  _Info^[_nAxisIndex].nErrorId      := 0;
  _eResultOld                       := _eResult;
END_IF
//-----------------------------------------------------------------------------
// encoder type (enum)
//-----------------------------------------------------------------------------
_State^[_nAxisIndex].eAxisEncoder   := EncoderType;
//-----------------------------------------------------------------------------
// Check ControlLoop
//-----------------------------------------------------------------------------
IF _AxisRef.Status.ControlLoopClosed
THEN
  _Info^[_nAxisIndex].bEnabled      := TRUE;
ELSE
  _Info^[_nAxisIndex].bEnabled      := FALSE;
END_IF
//-----------------------------------------------------------------------------
_Info^[_nAxisIndex].bStandstill     := _AxisRef.Status.NotMoving;
//-----------------------------------------------------------------------------
_Info^[_nAxisIndex].rActPos         := _AxisRef.NcToPlc.ActPos;
_Info^[_nAxisIndex].rActVelo        := _AxisRef.NcToPlc.ActVelo;
_Info^[_nAxisIndex].rPosDiff        := _AxisRef.NcToPlc.PosDiff;
//-----------------------------------------------------------------------------
IF (_Info^[_nAxisIndex].rActPos < _Data^[_nAxisIndex].rSetPos + _rTargetWindow) AND
   (_Info^[_nAxisIndex].rActPos > _Data^[_nAxisIndex].rSetPos - _rTargetWindow) AND
    _Info^[_nAxisIndex].bStandstill
THEN
  _Info^[_nAxisIndex].bInTarget     := TRUE;
ELSE
  _Info^[_nAxisIndex].bInTarget     := FALSE;
END_IF
//-----------------------------------------------------------------------------
// copy CoupleState from axis
//-----------------------------------------------------------------------------
_Info^[_nAxisIndex].dwCoupleState   := _AxisRef.NcToPlc.CoupleState;
//-----------------------------------------------------------------------------
//-----------------------------------------------------------------------------
// copy NC AxisId from axis
//-----------------------------------------------------------------------------
_Info^[_nAxisIndex].nNcAxisId       := _AxisRef.NcToPlc.AxisId;
//-----------------------------------------------------------------------------

PROPERTY Axes : reference TO ARRAY[1..PLC_CONSTANT.MAX_AXIS] OF AXIS_REF
SET
_Axes := Axes;
END_SET
END_PROPERTY

METHOD AxisBufferPos : E_PROGRESS
VAR_INPUT
  Enable            : BOOL;
  Data              : ST_MOVE_DATA;
END_VAR
VAR_INST
  _BufferMode       : Tc2_MC2.MC_BufferMode;
  _eres,
  _eState           : E_PROGRESS;
END_VAR
IF NOT Check() THEN AxisBufferPos := E_PROGRESS.ERROR; RETURN; END_IF
IF NOT Enable THEN _eState := E_PROGRESS.INIT; END_IF

CASE _eState
OF
  E_PROGRESS.INIT:
    IF Enable 
    THEN
      _eState       := E_PROGRESS.BUSY;
    END_IF
END_CASE
CASE _eState
OF
  E_PROGRESS.BUSY:
    _eState         := E_PROGRESS.WORKING;
    _BufferMode     := _MotionOptions^[_nAxisIndex].eBufferMode;
    _eres           := MovePosBuffer(
                                  Enable      := FALSE, 
                                  Position    := Data.rSetPos, 
                                  Vel         := Data.rSetVelo, 
                                  Acc         := Data.rAcc, 
                                  Dec         := Data.rDec, 
                                  Jerk        := Data.rJerk, 
                                  BufferMode  := _BufferMode);
END_CASE
CASE _eState
OF
  E_PROGRESS.WORKING:
    _BufferMode     := _MotionOptions^[_nAxisIndex].eBufferMode;
    AxisBufferPos   := _eres  
                    := MovePosBuffer(
                                  Enable      := TRUE, 
                                  Position    := Data.rSetPos, 
                                  Vel         := Data.rSetVelo, 
                                  Acc         := Data.rAcc, 
                                  Dec         := Data.rDec, 
                                  Jerk        := Data.rJerk, 
                                  BufferMode  := _BufferMode);
    IF (_eres = E_PROGRESS.ERROR)
    THEN
      _eState       := E_PROGRESS.ERROR;

    ELSIF (_Ctrl^[_nAxisIndex].eProgress = E_PROGRESS.DONE)
    THEN
      // when Ctrl decides to leave; make finishing move and be done
      _eState       := E_PROGRESS.DONE;
    END_IF
END_CASE
CASE _eState
OF
  E_PROGRESS.ERROR,
  E_PROGRESS.DONE:
    _eres           := MovePosBuffer(
                                  Enable      := FALSE, 
                                  Position    := Data.rSetPos, 
                                  Vel         := Data.rSetVelo, 
                                  Acc         := Data.rAcc, 
                                  Dec         := Data.rDec, 
                                  Jerk        := Data.rJerk, 
                                  BufferMode  := _BufferMode);

    AxisBufferPos   := _eState;
END_CASE
END_METHOD

METHOD AxisBufferVelo : E_PROGRESS
VAR_INPUT
  Enable            : BOOL;
  Data              : ST_MOVE_DATA;
END_VAR
VAR_INST
  _BufferMode       : Tc2_MC2.MC_BufferMode;
  _eres,
  _eState           : E_PROGRESS;
END_VAR
IF NOT Check() THEN AxisBufferVelo := E_PROGRESS.ERROR; RETURN; END_IF
IF NOT Enable THEN _eState := E_PROGRESS.INIT; END_IF

CASE _eState
OF
  E_PROGRESS.INIT:
    IF Enable 
    THEN
      _eState       := E_PROGRESS.BUSY;
    END_IF
END_CASE
CASE _eState
OF
  E_PROGRESS.BUSY:
    _eState         := E_PROGRESS.WORKING;
    _BufferMode     := _MotionOptions^[_nAxisIndex].eBufferMode;
    _eres           := MoveVeloBuffer(
                                  Enable      := FALSE, 
                                  Velocity    := Data.rSetVelo, 
                                  Acc         := Data.rAcc, 
                                  Dec         := Data.rDec, 
                                  Jerk        := Data.rJerk, 
                                  BufferMode  := _BufferMode);

END_CASE
CASE _eState
OF
  E_PROGRESS.WORKING:
    _BufferMode     := _MotionOptions^[_nAxisIndex].eBufferMode;
    _eres           := MoveVeloBuffer(
                                  Enable      := TRUE, 
                                  Velocity    := Data.rSetVelo, 
                                  Acc         := Data.rAcc, 
                                  Dec         := Data.rDec, 
                                  Jerk        := Data.rJerk, 
                                  BufferMode  := _BufferMode);
    IF (_eres = E_PROGRESS.ERROR)
    THEN
      _eState := E_PROGRESS.ERROR;
                       MoveVeloBuffer(
                                  Enable      := FALSE, 
                                  Velocity    := Data.rSetVelo, 
                                  Acc         := Data.rAcc, 
                                  Dec         := Data.rDec, 
                                  Jerk        := Data.rJerk, 
                                  BufferMode  := _BufferMode);

    ELSIF (_Ctrl^[_nAxisIndex].eProgress = E_PROGRESS.DONE)
    THEN
      // when Ctrl decides to leave; make finishing move and be done
      _eState       := E_PROGRESS.FINISHING;
    END_IF
END_CASE
CASE _eState
OF
  E_PROGRESS.FINISHING:
    _eState         := E_PROGRESS.DONE;
    _eres           := MoveVeloBuffer(
                                  Enable      := FALSE, 
                                  Velocity    := Data.rSetVelo, 
                                  Acc         := Data.rAcc, 
                                  Dec         := Data.rDec, 
                                  Jerk        := Data.rJerk, 
                                  BufferMode  := _BufferMode);
END_CASE

AxisBufferVelo      := _eState;
END_METHOD

PROPERTY AxisCtrl : pointer to ARRAY[1..PLC_CONSTANT.MAX_AXIS] OF st_axis_ctrl
SET
_Ctrl := AxisCtrl;
END_SET
END_PROPERTY

PROPERTY AxisData : pointer to ARRAY[1..PLC_CONSTANT.MAX_AXIS] OF st_move_data
SET
_Data := AxisData;
END_SET
END_PROPERTY

METHOD AxisDisable : E_PROGRESS
VAR_INPUT
  Execute           : BOOL;
END_VAR
VAR_INST
  _eState,
  _eResult          : E_PROGRESS;
  _rValue           : LREAL;
  _udiErr           : UDINT;
  _stMsg            : ST_Message;


END_VAR
IF NOT Check() THEN AxisDisable := E_PROGRESS.ERROR; RETURN; END_IF
IF NOT Execute THEN _eState := E_PROGRESS.INIT; END_IF

CASE _eState
OF
  E_PROGRESS.INIT:
    IF Execute 
    THEN
      memset(ADR(_stMsg),0,SIZEOF(_stMsg));
      _udiErr                       := 0;
      _rValue                       := 0;
      _eState                       := E_PROGRESS.BUSY;
    END_IF
END_CASE
CASE _eState
OF
  E_PROGRESS.BUSY:
    _eResult                        := Disable(FALSE);
    _eState                         := E_PROGRESS.WAITING;
END_CASE
CASE _eState
OF
  E_PROGRESS.WAITING:
    _eResult                        := Disable(TRUE);

    IF (_eResult = E_PROGRESS.DONE)
    THEN
      _eState                       := E_PROGRESS.WORKING;
    END_IF
END_CASE
CASE _eState
OF
  E_PROGRESS.WORKING:
    _eState                         := E_PROGRESS.DONE;
END_CASE

AxisDisable := _eState;
END_METHOD

METHOD AxisEnable : E_PROGRESS
VAR_INPUT
  Execute           : BOOL;
END_VAR
VAR_INST
  _eState,
  _eResult          : E_PROGRESS;
  _rValue           : LREAL;
  _udiErr           : UDINT;
  _stMsg            : ST_Message;


END_VAR
IF NOT Check() THEN AxisEnable := E_PROGRESS.ERROR; RETURN; END_IF
IF NOT Execute THEN _eState := E_PROGRESS.INIT; END_IF

CASE _eState
OF
  E_PROGRESS.INIT:
    IF Execute 
    THEN
      memset(ADR(_stMsg),0,SIZEOF(_stMsg));
      _udiErr                       := 0;
      _rValue                       := 0;
      _eState                       := E_PROGRESS.BUSY;
    END_IF
END_CASE
CASE _eState
OF
  E_PROGRESS.BUSY:
    _eResult                        := Enable(FALSE);
    _eState                         := E_PROGRESS.WAITING;
END_CASE
CASE _eState
OF
  E_PROGRESS.WAITING:
    _eResult                        := Enable(TRUE);

    IF (_eResult = E_PROGRESS.DONE)
    THEN
      _eState                       := E_PROGRESS.WORKING;
    END_IF
END_CASE
CASE _eState
OF
  E_PROGRESS.WORKING:
    _eState                         := E_PROGRESS.DONE;
END_CASE

AxisEnable := _eState;
END_METHOD

METHOD AxisGearIn : E_PROGRESS
VAR_INPUT
  Execute           : BOOL;
END_VAR
VAR_INST
  _eState           : E_PROGRESS;
  _rValue           : LREAL;
  _nErr,
  _nMasterIndex,
  _nMasterNcId      : UDINT;
  _stMsg            : ST_Message;


END_VAR
IF NOT Check() THEN AxisGearIn := E_PROGRESS.ERROR; RETURN; END_IF
IF NOT Execute THEN _eState := E_PROGRESS.INIT; END_IF

CASE _eState
OF
  E_PROGRESS.INIT:
    IF Execute 
    THEN
      memset(ADR(_stMsg),0,SIZEOF(_stMsg));
      _nMasterNcId                  :=
      _nMasterIndex                 :=
      _nErr                         := 0;
      _rValue                       := 0;

      IF NOT (_GearInParameter^[_nAxisIndex].nAxisIndexMaster[1] > 0) OR
         NOT (_GearInParameter^[_nAxisIndex].nAxisIndexMaster[1] < MAX_AXIS+1)
      THEN
        _nMasterIndex               := _GearInParameter^[_nAxisIndex].nAxisIndexMaster[1];

        _stMsg.eType                := E_MessageType.eMessageError;
        _stMsg.eDevice              := e_Device.Axis + TO_UINT(_AxisRef.NcToPlc.AxisId);
        _stMsg.eSubdevice           := e_Subdevice.fbGearIn;
        _stMsg.iErrorNumber         := 
        _nErr                       := 666;

        _stMsg.sText                := concat('_GearInParameter[', TO_STRING(_nAxisIndex));
        _stMsg.sText                := concat(_stMsg.sText,    '].nAxisIndexMaster[1] out of range: ');
        _stMsg.sText                := concat(_stMsg.sText, TO_STRING(_nMasterIndex));

        f_MessageSet(_stMsg);

        _eState                     := E_PROGRESS.ERROR;

      ELSE
        _eState                     := E_PROGRESS.BUSY;

        _nMasterIndex               := _GearInParameter^[_nAxisIndex].nAxisIndexMaster[1];
        _nMasterNcId                := _Info^[_nMasterIndex].nNcAxisId;

        _stMsg.eType                := E_MessageType.eMessageInfo;
        _stMsg.eDevice              := e_Device.Axis + TO_UINT(_AxisRef.NcToPlc.AxisId);
        _stMsg.eSubdevice           := e_Subdevice.fbGearIn;
        _stMsg.iErrorNumber         := 0;
  
        _stMsg.sText                := concat('GearIn BUSY: ', TO_STRING(_nMasterIndex));
        f_MessageSet(_stMsg);
      END_IF
    END_IF
END_CASE
CASE _eState
OF
  E_PROGRESS.BUSY:
    _eState                         := E_PROGRESS.STARTUP;
    _fbGearIn(
              Master                := _Axes[_nMasterIndex], 
              Slave                 := _AxisRef, 
              Execute               := FALSE, 
              RatioNumerator        := _GearInParameter^[_nAxisIndex].rGearRatio[1], 
              RatioDenominator      := 1, 
              Acceleration          := _GearInParameter^[_nAxisIndex].Acceleration, 
              Deceleration          := _GearInParameter^[_nAxisIndex].Deceleration, 
              Jerk                  := _GearInParameter^[_nAxisIndex].Jerk);
END_CASE
CASE _eState
OF
  E_PROGRESS.STARTUP:
    _fbGearIn(
              Master                := _Axes[_nMasterIndex], 
              Slave                 := _AxisRef, 
              Execute               := TRUE, 
              RatioNumerator        := _GearInParameter^[_nAxisIndex].rGearRatio[1], 
              RatioDenominator      := 1, 
              Acceleration          := _GearInParameter^[_nAxisIndex].Acceleration, 
              Deceleration          := _GearInParameter^[_nAxisIndex].Deceleration, 
              Jerk                  := _GearInParameter^[_nAxisIndex].Jerk);

    IF (_fbGearIn.Error)
    THEN
      _nErr                         := _fbGearIn.ErrorID;

      _stMsg.eType                  := E_MessageType.eMessageError;
      _stMsg.eDevice                := e_Device.Axis + TO_UINT(_AxisRef.NcToPlc.AxisId);
      _stMsg.eSubdevice             := e_Subdevice.fbGearIn;
      _stMsg.iErrorNumber           := _nErr;

      _stMsg.sText                  := concat('GearIn ERROR: ', TO_STRING(_nMasterIndex));
      f_MessageSet(_stMsg);
      _eState                       := E_PROGRESS.ERROR;

    ELSIF (_fbGearIn.InGear)
    THEN
      _eState                       := E_PROGRESS.READY;
    END_IF
END_CASE
CASE _eState
OF
  E_PROGRESS.READY:
    _eState                         := E_PROGRESS.DONE;

    _stMsg.eType                    := E_MessageType.eMessageInfo;
    _stMsg.eDevice                  := e_Device.Axis + TO_UINT(_AxisRef.NcToPlc.AxisId);
    _stMsg.eSubdevice               := e_Subdevice.fbGearIn;
    _stMsg.iErrorNumber             := 0;

    _stMsg.sText                    := concat('GearIn done: ', TO_STRING(_nMasterIndex));
    f_MessageSet(_stMsg);
END_CASE
CASE _eState
OF
  E_PROGRESS.DONE,
  E_PROGRESS.ERROR:
    _fbGearIn(
              Master                := _Axes[_nMasterIndex], 
              Slave                 := _AxisRef, 
              Execute               := FALSE);
END_CASE

AxisGearIn                          := _eState;
END_METHOD

METHOD AxisGearInMultiMaster : E_PROGRESS
VAR_INPUT
  Execute           : BOOL;
END_VAR
VAR_INST
  _eState           : E_PROGRESS;
  _rValue           : LREAL;
  _nAx,
  _nErr             : UDINT;

  _nMasterIndex,
  _nMasterNcId      : ARRAY[1..4] OF UDINT;

  _stOptions        : Tc2_MC2.ST_GearInMultiMasterOptions;
  _nSyncMode        : int;

  _stMsg            : ST_Message;


END_VAR
IF NOT Check() THEN AxisGearInMultiMaster := E_PROGRESS.ERROR; RETURN; END_IF
IF NOT Execute THEN _eState := E_PROGRESS.INIT; END_IF

CASE _eState
OF
  E_PROGRESS.INIT:
    IF Execute 
    THEN
      memset(ADR(_stMsg),0,SIZEOF(_stMsg));
      memset(ADR(_nMasterNcId), 0,SIZEOF(_nMasterNcId));
      memset(ADR(_nMasterIndex),0,SIZEOF(_nMasterIndex));
      memset(ADR(_stOptions),   0,SIZEOF(_stOptions));
      _nErr                           := 0;
      _rValue                         := 0;

      IF NOT (_GearInParameter^[_nAxisIndex].nAxisIndexMaster[1] > 0) OR
         NOT (_GearInParameter^[_nAxisIndex].nAxisIndexMaster[1] <= MAX_AXIS)
      THEN
        _nMasterIndex[1]              := _GearInParameter^[_nAxisIndex].nAxisIndexMaster[1];

        _stMsg.eType                  := E_MessageType.eMessageError;
        _stMsg.eDevice                := e_Device.Axis + TO_UINT(_AxisRef.NcToPlc.AxisId);
        _stMsg.eSubdevice             := e_Subdevice.fbGearInMultiMaster;
        _stMsg.iErrorNumber           := 
        _nErr                         := 666;

        _stMsg.sText                  := concat('_GearInParameter[', TO_STRING(_nAxisIndex));
        _stMsg.sText                  := concat(_stMsg.sText,    '].nAxisIndexMaster[1] out of range: ');
        _stMsg.sText                  := concat(_stMsg.sText, TO_STRING(_nMasterIndex[1]));
        f_MessageSet(_stMsg);

        _eState                       := E_PROGRESS.ERROR;

      ELSE
        _eState                       := E_PROGRESS.BUSY;

        _stOptions.AdvancedSlaveDynamics  := _GearInParameter^[_nAxisIndex].bAdvancedSlaveDynamics;
        _nSyncMode                        := _GearInParameter^[_nAxisIndex].nMultiMasterSyncMode;

        _nMasterIndex[1]              := _GearInParameter^[_nAxisIndex].nAxisIndexMaster[1];
        _nMasterNcId[1]               := _Info^[_nMasterIndex[1]].nNcAxisId;
        memcpy(ADR(_stOptions.SyncMode), ADR(_nSyncMode), SIZEOF(_stOptions.SyncMode));

        _fbGearInMultiMaster.Master1  := _Axes[_nMasterIndex[1]];   // assign AXIS_REF of master

        _stMsg.eType                  := E_MessageType.eMessageInfo;
        _stMsg.eDevice                := e_Device.Axis + TO_UINT(_AxisRef.NcToPlc.AxisId);
        _stMsg.eSubdevice             := e_Subdevice.fbGearInMultiMaster;
        _stMsg.iErrorNumber           := _eState;

        _stMsg.sText                  := concat('_GearInParameter[', TO_STRING(_nAxisIndex));
        _stMsg.sText                  := concat(_stMsg.sText,    '] MultiMaster check: ');
        _stMsg.sText                  := concat(_stMsg.sText, TO_STRING(_nMasterIndex[1]));
        f_MessageSet(_stMsg);

        _nAx                          := 2; // next master index to check
      END_IF
    END_IF
END_CASE
CASE _eState
OF
  E_PROGRESS.BUSY:
    IF NOT (_GearInParameter^[_nAxisIndex].nAxisIndexMaster[_nAx] > 0) OR
       NOT (_GearInParameter^[_nAxisIndex].nAxisIndexMaster[_nAx] < MAX_AXIS+1)
    THEN
      // next entry not valid
      // Master1 is already checked --> let's get ready
      _eState                         := E_PROGRESS.READY;
    ELSE
      _eState                         := E_PROGRESS.STARTUP;

      _nMasterIndex[_nAx]             := _GearInParameter^[_nAxisIndex].nAxisIndexMaster[_nAx];
      _nMasterNcId [_nAx]             := _Info^[_nMasterIndex[_nAx]].nNcAxisId;

      _stMsg.eType                    := E_MessageType.eMessageInfo;
      _stMsg.eDevice                  := e_Device.Axis + TO_UINT(_AxisRef.NcToPlc.AxisId);
      _stMsg.eSubdevice               := e_Subdevice.fbGearInMultiMaster;
      _stMsg.iErrorNumber             := _eState;

